(* CoDeSys 2.3.9.41 project: VOS_Vorkuta_ASU_3_osmos_2.pro *)
(* Libraries: PID_Regulators.lib 6.11.19 15:29:27, Util.lib 18.5.10 15:14:28, STANDARD.LIB 4.10.05 11:14:46, IECSFC.LIB 13.4.06 15:51:28, GermesLib_1_4.lib 25.4.21 16:11:00, SYSLIBTIME.LIB 6.11.19 15:29:28, ANALYZATION.LIB 5.10.99 09:05:06 *)

(* PLC configuration (modules and I/O channels)
Fast discrete inputs [I_SIMPLE_INPUT] node 0, in %IB0 out %QB0 {ChannellName = Fast discrete inputs; Filtrationtime = 10000}
  DD1_DI_1 AT %IX0.0 [BitInput] Авария насоса Р03.01/01 {ChannellName = Enter name}
  DD1_DI_2 AT %IX0.1 [BitInput] Авария насоса Р03.01/02 {ChannellName = Enter name}
  DD1_DI_3 AT %IX0.2 [BitInput] эк.манометр PIS03.01/01 после насоса Р03.01/01 {ChannellName = Enter name}
  DD1_DI_4 AT %IX0.3 [BitInput] эк.манометр PIS03.01/02 после насоса Р03.01/02 {ChannellName = Enter name}
Discrete inputs [ID130] node 1, in %IB1 out %QB1 {ChannellName = Discrete inputs; Filtrationtime_GeneralINP = 10; PinCount = 12; Visibility = No}
  AT %IB1.0 [ByteInput] 8 discrete inputs {ChannellName = Enter name}
  AT %IB1.1 [ByteInput] 4 discrete inputs {ChannellName = Enter name}
Fast discrete outputs [OWEN_ID570] node 2, in %IB2 out %QB2 {ChannellName = Fast discrete outputs; SafeValueBool = FALSE; SafeValueBool = FALSE; SafeValueBool = FALSE; SafeValueBool = FALSE; Visibility = No}
  DD1_DO_1 AT %QX2.0 [BitOutput] Fast discrete output 1 {ChannellName = Enter name}
  DD1_DO_2 AT %QX2.1 [BitOutput] Fast discrete output 2 {ChannellName = Enter name}
  DD1_DO_3 AT %QX2.2 [BitOutput] Fast discrete output 3 {ChannellName = Enter name}
  DD1_DO_4 AT %QX2.3 [BitOutput] Fast discrete output 4 {ChannellName = Enter name}
Discrete outputs [ID131] node 3, in %IB3 out %QB3 {ChannellName = Discrete outputs; SafeValueByte = 0; Visibility = No}
  AT %QB3.0 [ByteOutput] 8 discrete outputs {ChannellName = Enter name}
  AT %QB3.1 [ByteOutput] 8 discrete outputs {ChannellName = Enter name}
Fast analog inputs [ID125] node 4, in %IB4 out %QB4 {ChannellName = Fast analog inputs; Flt_Comm = 50Hz 2Por}
  DD1_AI_1 AT %IR4.0 [FloatInputP] резерв {ChannellName = Fast analog input; AIN_TYPE = 0-20 mA; Peak_Filtr = 200; Flt_Ch = Off; TauRC = 10; MinFV = 0; MaxFV = 20}
  DD1_AI_2 AT %IR4.1 [FloatInputP] датчик давления РТ03.01/01 {ChannellName = Fast analog input; AIN_TYPE = 0-20 mA; Peak_Filtr = 200; Flt_Ch = Off; TauRC = 10; MinFV = 0; MaxFV = 20}
  DD1_AI_3 AT %IR4.2 [FloatInputP] датчик давления РТ03.02/01 {ChannellName = Fast analog input; AIN_TYPE = 0-20 mA; Peak_Filtr = 200; Flt_Ch = Off; TauRC = 10; MinFV = 0; MaxFV = 20}
  DD1_AI_4 AT %IR4.3 [FloatInputP] датчик давления РТ03.03/01 {ChannellName = Fast analog input; AIN_TYPE = 0-20 mA; Peak_Filtr = 200; Flt_Ch = Off; TauRC = 10; MinFV = 0; MaxFV = 20}
  DD1_AI_5 AT %IR4.4 [FloatInputP] датчик давления РТ03.04/01 {ChannellName = Fast analog input; AIN_TYPE = 0-20 mA; Peak_Filtr = 200; Flt_Ch = Off; TauRC = 10; MinFV = 0; MaxFV = 20}
  DD1_AI_6 AT %IR4.5 [FloatInputP] кондуктомер QIT03.01/01 осн.осмос {ChannellName = Fast analog input; AIN_TYPE = 0-20 mA; Peak_Filtr = 200; Flt_Ch = Off; TauRC = 10; MinFV = 0; MaxFV = 20}
  DD1_AI_7 AT %IR4.6 [FloatInputP] расходомер FIT03.02/01 осн.осмос {ChannellName = Fast analog input; AIN_TYPE = 0-20 mA; Peak_Filtr = 200; Flt_Ch = Off; TauRC = 10; MinFV = 0; MaxFV = 20}
  DD1_AI_8 AT %IR4.7 [FloatInputP] расходомер FIT03.03/01 осн.осмос {ChannellName = Fast analog input; AIN_TYPE = 0-20 mA; Peak_Filtr = 200; Flt_Ch = Off; TauRC = 10; MinFV = 0; MaxFV = 20}
  AT %IW4.8 [WordInput] AI read time (10ms) {ChannellName = Enter name}
Analog outputs [ID126] node 5, in %IB5 out %QB5 {ChannellName = Analog outputs}
  DD1_AO_1 AT %QR5.0 [FloatOutputP] производительность осн.доз.насоса Р03.02/01 {ChannellName = Analog output; AOUT_TYPE = 4-20 mA; SafeValueREAL = 0.0}
  DD1_AO_2 AT %QR5.1 [FloatOutputP] производительность рез.доз.насоса Р03.02/02 {ChannellName = Analog output; AOUT_TYPE = 4-20 mA; SafeValueREAL = 0.0}
  DD1_AO_3 AT %QR5.2 [FloatOutputP] резерв {ChannellName = Analog output; AOUT_TYPE = 4-20 mA; SafeValueREAL = 0.0}
  DD1_AO_4 AT %QR5.3 [FloatOutputP] резерв {ChannellName = Analog output; AOUT_TYPE = 4-20 mA; SafeValueREAL = 0.0}
Special input [ID103] node 6, in %IB6 out %QB6 {ChannellName = Special input}
  AT %IX6.0 [BitInput] Special input {ChannellName = Enter name}
Special output [ID104] node 7, in %IB7 out %QB7 {ChannellName = Special output}
  AT %QX7.0 [BitOutput] Special output {ChannellName = Enter name}
ModBus (Master) [MODBUS_MASTER_ID450] node 8, in %IB8 out %QB8 {ChannellName = ModBus (Master); Visibility = No}
  AT %QD8.0 [DWordOutput] Last address {ChannellName = Enter name}
  AT %QW8.1 [WordOutput] Last error {ChannellName = Enter name}
  RS-485-1 [COM1_USART] node 0, in %IB8.0 out %QB8.0 {ChannellName = RS-485-1; CommunicationSpeed = 9600; Parity = NO PARITY CHECK; BitLength = 8 bits; StopLength = One stop bit; InterfaceType = RS485; FrameOriented = RTU; Timeout = 5; Visibility = No}
  Universal Modbus device [ID2000] node 1, in %IB8.1 out %QB8.1 {ChannellName = Universal Modbus device; ModuleIP = 10:0:0:223; ServiceTimeout = 150; TCPport = 502; NetMode = Serial; ModuleSlaveAddress = 11; RequestType = By poll time; PeriodOfService = 100; Visibility = No; RepeatCounter = 0; ByteSequence = Native}
    AT %QB8.1.0 [ComChannel] Command (0xff - Start) {ChannellName = Enter name}
    Real input module [ID2007] node 0, in %IB8.1.0 out %QB8.1.0 {ChannellName = float input module; ModbusAddress = 512; Command_read_regs = Read holding Registers  (0x03); Visibility = No}
      PT030102rawValue AT %QD8.1.0.0 [FloatOutput] {ChannellName = Enter name}
    Real input module [ID2007] node 1, in %IB8.1.1 out %QB8.1.1 {ChannellName = float input module; ModbusAddress = 514; Command_read_regs = Read holding Registers  (0x03); Visibility = No}
      PT030202rawValue AT %QD8.1.1.0 [FloatOutput] {ChannellName = Enter name}
    Real input module [ID2007] node 2, in %IB8.1.2 out %QB8.1.2 {ChannellName = float input module; ModbusAddress = 516; Command_read_regs = Read holding Registers  (0x03); Visibility = No}
      PT030302rawValue AT %QD8.1.2.0 [FloatOutput] {ChannellName = Enter name}
    Real input module [ID2007] node 3, in %IB8.1.3 out %QB8.1.3 {ChannellName = float input module; ModbusAddress = 518; Command_read_regs = Read holding Registers  (0x03); Visibility = No}
      PT030402rawValue AT %QD8.1.3.0 [FloatOutput] {ChannellName = Enter name}
    Real input module [ID2007] node 4, in %IB8.1.4 out %QB8.1.4 {ChannellName = float input module; ModbusAddress = 520; Command_read_regs = Read holding Registers  (0x03); Visibility = No}
      QIT030102rawValue AT %QD8.1.4.0 [FloatOutput] {ChannellName = Enter name}
    Real input module [ID2007] node 5, in %IB8.1.5 out %QB8.1.5 {ChannellName = float input module; ModbusAddress = 522; Command_read_regs = Read holding Registers  (0x03); Visibility = No}
      FIT030202rawValue AT %QD8.1.5.0 [FloatOutput] {ChannellName = Enter name}
    Real input module [ID2007] node 6, in %IB8.1.6 out %QB8.1.6 {ChannellName = float input module; ModbusAddress = 524; Command_read_regs = Read holding Registers  (0x03); Visibility = No}
      FIT030302rawValue AT %QD8.1.6.0 [FloatOutput] {ChannellName = Enter name}
    Real input module [ID2007] node 7, in %IB8.1.7 out %QB8.1.7 {ChannellName = float input module; ModbusAddress = 526; Command_read_regs = Read holding Registers  (0x03); Visibility = No}
      FIT030101rawValue AT %QD8.1.7.0 [FloatOutput] {ChannellName = Enter name}
    Register input module [ID2003] node 8, in %IB8.1.8 out %QB8.1.8 {ChannellName = Register input module; ModbusAddress = 529; Command_read_regs = Read input registers  (0x04); Visibility = No}
      DI_bit_mask_DD2 AT %QW8.1.8.0 [WordOutput] {ChannellName = Enter name}
    Register input module [ID2003] node 9, in %IB8.1.9 out %QB8.1.9 {ChannellName = Register input module; ModbusAddress = 532; Command_read_regs = Read input registers  (0x04); Visibility = No}
      stat_word_P030601_PLC AT %QW8.1.9.0 [WordOutput] {ChannellName = Enter name}
    Register input module [ID2003] node 10, in %IB8.1.10 out %QB8.1.10 {ChannellName = Register input module; ModbusAddress = 535; Command_read_regs = Read input registers  (0x04); Visibility = No}
      stat_word_P030602_PLC AT %QW8.1.10.0 [WordOutput] {ChannellName = Enter name}
  Universal Modbus device [ID2000] node 2, in %IB8.2 out %QB8.2 {ChannellName = Universal Modbus device; ModuleIP = 10:0:0:223; ServiceTimeout = 150; TCPport = 502; NetMode = Serial; ModuleSlaveAddress = 1; RequestType = By value change; PeriodOfService = 100; Visibility = No; RepeatCounter = 0; ByteSequence = Native}
    AT %QB8.2.0 [ComChannel] Command (0xff - Start) {ChannellName = Enter name}
    Register output module [ID2004] node 0, in %IB8.2.0 out %QB8.2.0 {ChannellName = Register; ModbusAddress = 528; Command_write_one_reg = Write multiple registers(0x10); Visibility = No}
      DO_bit_mask_DD2 AT %QW8.2.0.0 [WordOutput] {ChannellName = Enter name}
    Register output module [ID2004] node 1, in %IB8.2.1 out %QB8.2.1 {ChannellName = Register; ModbusAddress = 530; Command_write_one_reg = Write multiple registers(0x10); Visibility = No}
      com_word_P030601_PLC AT %QW8.2.1.0 [WordOutput] {ChannellName = Enter name}
    Register output module [ID2004] node 2, in %IB8.2.2 out %QB8.2.2 {ChannellName = Register; ModbusAddress = 531; Command_write_one_reg = Write multiple registers(0x10); Visibility = No}
      set_freq_P030601_PLC AT %QW8.2.2.0 [WordOutput] {ChannellName = Enter name}
    Register output module [ID2004] node 3, in %IB8.2.3 out %QB8.2.3 {ChannellName = Register; ModbusAddress = 533; Command_write_one_reg = Write multiple registers(0x10); Visibility = No}
      com_word_P030602_PLC AT %QW8.2.3.0 [WordOutput] {ChannellName = Enter name}
    Register output module [ID2004] node 4, in %IB8.2.4 out %QB8.2.4 {ChannellName = Register; ModbusAddress = 534; Command_write_one_reg = Write multiple registers(0x10); Visibility = No}
      set_freq_P030602_PLC AT %QW8.2.4.0 [WordOutput] {ChannellName = Enter name}
ModBus (Master) [MODBUS_MASTER_ID450] node 9, in %IB9 out %QB9 {ChannellName = ModBus (Master); Visibility = No}
  AT %QD9.0 [DWordOutput] Last address {ChannellName = Enter name}
  AT %QW9.1 [WordOutput] Last error {ChannellName = Enter name}
  RS-232 [COM2_USART] node 0, in %IB9.0 out %QB9.0 {ChannellName = RS-232; CommunicationSpeed = 115200; Parity = NO PARITY CHECK; BitLength = 8 bits; StopLength = One stop bit; InterfaceType = RS232; FrameOriented = RTU; Timeout = 5; Visibility = No}
  Universal Modbus device [ID2000] node 1, in %IB9.1 out %QB9.1 {ChannellName = Universal Modbus device; ModuleIP = 10:0:0:223; ServiceTimeout = 150; TCPport = 502; NetMode = Serial; ModuleSlaveAddress = 1; RequestType = By poll time; PeriodOfService = 50; Visibility = No; RepeatCounter = 0; ByteSequence = Native}
    AT %QB9.1.0 [ComChannel] Command (0xff - Start) {ChannellName = Enter name}
    Register input module [ID2003] node 0, in %IB9.1.0 out %QB9.1.0 {ChannellName = Register input module; ModbusAddress = 10256; Command_read_regs = Read holding Registers  (0x03); Visibility = No}
      PANsetWordP0301 AT %QW9.1.0.0 [WordOutput] {ChannellName = Enter name}
    Register input module [ID2003] node 1, in %IB9.1.1 out %QB9.1.1 {ChannellName = Register input module; ModbusAddress = 10257; Command_read_regs = Read holding Registers  (0x03); Visibility = No}
      PANsetWordP0302 AT %QW9.1.1.0 [WordOutput] {ChannellName = Enter name}
PAN_FIT0301maxValue AT %QD9.1.2.0 [FloatOutput] {ChannellName = Enter name}
Real input module [ID2007] node 3, in %IB9.1.3 out %QB9.1.3 {ChannellName = float input module; ModbusAddress = 10260; Command_read_regs = Read holding Registers  (0x03); Visibility = No}
  PANsetMaxPumpDosingValueP0302 AT %QD9.1.3.0 [FloatOutput] {ChannellName = Enter name}
Real input module [ID2007] node 4, in %IB9.1.4 out %QB9.1.4 {ChannellName = float input module; ModbusAddress = 10262; Command_read_regs = Read holding Registers  (0x03); Visibility = No}
  PANsetKoeffPropotrionalityP0302 AT %QD9.1.4.0 [FloatOutput] {ChannellName = Enter name}
Register input module [ID2003] node 5, in %IB9.1.5 out %QB9.1.5 {ChannellName = Register input module; ModbusAddress = 10264; Command_read_regs = Read holding Registers  (0x03); Visibility = No}
  PAN_CHECKING_DELAY_TIME AT %QW9.1.5.0 [WordOutput] {ChannellName = Enter name}
Register input module [ID2003] node 6, in %IB9.1.6 out %QB9.1.6 {ChannellName = Register input module; ModbusAddress = 10265; Command_read_regs = Read holding Registers  (0x03); Visibility = No}
  PAN_DELAY_REPEATED_START_SEC AT %QW9.1.6.0 [WordOutput] {ChannellName = Enter name}
Register input module [ID2003] node 7, in %IB9.1.7 out %QB9.1.7 {ChannellName = Register input module; ModbusAddress = 10266; Command_read_regs = Read holding Registers  (0x03); Visibility = No}
  PAN_DELAY_TO_OFF_VALVE AT %QW9.1.7.0 [WordOutput] {ChannellName = Enter name}
Register input module [ID2003] node 8, in %IB9.1.8 out %QB9.1.8 {ChannellName = Register input module; ModbusAddress = 10267; Command_read_regs = Read holding Registers  (0x03); Visibility = No}
  PAN_DELAY_TO_CHECK_PT0301 AT %QW9.1.8.0 [WordOutput] {ChannellName = Enter name}
Register input module [ID2003] node 9, in %IB9.1.9 out %QB9.1.9 {ChannellName = Register input module; ModbusAddress = 10268; Command_read_regs = Read holding Registers  (0x03); Visibility = No}
  PAN_DELAY_TO_SWITCH_VALVE AT %QW9.1.9.0 [WordOutput] {ChannellName = Enter name}
Register input module [ID2003] node 10, in %IB9.1.10 out %QB9.1.10 {ChannellName = Register input module; ModbusAddress = 10269; Command_read_regs = Read holding Registers  (0x03); Visibility = No}
  PAN_DELAY_TO_CLOSE_VALVE AT %QW9.1.10.0 [WordOutput] {ChannellName = Enter name}
Real input module [ID2007] node 11, in %IB9.1.11 out %QB9.1.11 {ChannellName = float input module; ModbusAddress = 10276; Command_read_regs = Read holding Registers  (0x03); Visibility = No}
  PAN_FIT030201maxValue AT %QD9.1.11.0 [FloatOutput] {ChannellName = Enter name}
Real input module [ID2007] node 12, in %IB9.1.12 out %QB9.1.12 {ChannellName = float input module; ModbusAddress = 10278; Command_read_regs = Read holding Registers  (0x03); Visibility = No}
  PAN_FIT030301maxValue AT %QD9.1.12.0 [FloatOutput] {ChannellName = Enter name}
Real input module [ID2007] node 13, in %IB9.1.13 out %QB9.1.13 {ChannellName = float input module; ModbusAddress = 10280; Command_read_regs = Read holding Registers  (0x03); Visibility = No}
  PAN_FIT030202maxValue AT %QD9.1.13.0 [FloatOutput] {ChannellName = Enter name}
Real input module [ID2007] node 14, in %IB9.1.14 out %QB9.1.14 {ChannellName = float input module; ModbusAddress = 10282; Command_read_regs = Read holding Registers  (0x03); Visibility = No}
  PAN_FIT030302maxValue AT %QD9.1.14.0 [FloatOutput] {ChannellName = Enter name}
Real input module [ID2007] node 15, in %IB9.1.15 out %QB9.1.15 {ChannellName = float input module; ModbusAddress = 10284; Command_read_regs = Read holding Registers  (0x03); Visibility = No}
  PAN_QIT030101maxValue AT %QD9.1.15.0 [FloatOutput] {ChannellName = Enter name}
Real input module [ID2007] node 16, in %IB9.1.16 out %QB9.1.16 {ChannellName = float input module; ModbusAddress = 10286; Command_read_regs = Read holding Registers  (0x03); Visibility = No}
  PAN_QIT030102maxValue AT %QD9.1.16.0 [FloatOutput] {ChannellName = Enter name}
Real input module [ID2007] node 17, in %IB9.1.17 out %QB9.1.17 {ChannellName = float input module; ModbusAddress = 10288; Command_read_regs = Read holding Registers  (0x03); Visibility = No}
  PAN_PT030101maxValue AT %QD9.1.17.0 [FloatOutput] {ChannellName = Enter name}
Real input module [ID2007] node 18, in %IB9.1.18 out %QB9.1.18 {ChannellName = float input module; ModbusAddress = 10290; Command_read_regs = Read holding Registers  (0x03); Visibility = No}
  PAN_PT030201maxValue AT %QD9.1.18.0 [FloatOutput] {ChannellName = Enter name}
Real input module [ID2007] node 19, in %IB9.1.19 out %QB9.1.19 {ChannellName = float input module; ModbusAddress = 10292; Command_read_regs = Read holding Registers  (0x03); Visibility = No}
  PAN_PT030301maxValue AT %QD9.1.19.0 [FloatOutput] {ChannellName = Enter name}
Real input module [ID2007] node 20, in %IB9.1.20 out %QB9.1.20 {ChannellName = float input module; ModbusAddress = 10294; Command_read_regs = Read holding Registers  (0x03); Visibility = No}
  PAN_PT030401maxValue AT %QD9.1.20.0 [FloatOutput] {ChannellName = Enter name}
Real input module [ID2007] node 21, in %IB9.1.21 out %QB9.1.21 {ChannellName = float input module; ModbusAddress = 10296; Command_read_regs = Read holding Registers  (0x03); Visibility = No}
  PAN_PT030102maxValue AT %QD9.1.21.0 [FloatOutput] {ChannellName = Enter name}
Real input module [ID2007] node 22, in %IB9.1.22 out %QB9.1.22 {ChannellName = float input module; ModbusAddress = 10298; Command_read_regs = Read holding Registers  (0x03); Visibility = No}
  PAN_PT030202maxValue AT %QD9.1.22.0 [FloatOutput] {ChannellName = Enter name}
Real input module [ID2007] node 23, in %IB9.1.23 out %QB9.1.23 {ChannellName = float input module; ModbusAddress = 10300; Command_read_regs = Read holding Registers  (0x03); Visibility = No}
  PAN_PT030302maxValue AT %QD9.1.23.0 [FloatOutput] {ChannellName = Enter name}
Real input module [ID2007] node 24, in %IB9.1.24 out %QB9.1.24 {ChannellName = float input module; ModbusAddress = 10302; Command_read_regs = Read holding Registers  (0x03); Visibility = No}
  PAN_PT030402maxValue AT %QD9.1.24.0 [FloatOutput] {ChannellName = Enter name}
PANsetWordOsmos AT %QW9.1.25.0 [WordOutput] {ChannellName = Enter name}
Real input module [ID2007] node 26, in %IB9.1.26 out %QB9.1.26 {ChannellName = float input module; ModbusAddress = 10306; Command_read_regs = Read holding Registers  (0x03); Visibility = No}
  PAN_PT0301startValue AT %QD9.1.26.0 [FloatOutput] {ChannellName = Enter name}
Real input module [ID2007] node 27, in %IB9.1.27 out %QB9.1.27 {ChannellName = float input module; ModbusAddress = 10308; Command_read_regs = Read holding Registers  (0x03); Visibility = No}
  PAN_FIT0303setValue AT %QD9.1.27.0 [FloatOutput] {ChannellName = Enter name}
Real input module [ID2007] node 28, in %IB9.1.28 out %QB9.1.28 {ChannellName = float input module; ModbusAddress = 10310; Command_read_regs = Read holding Registers  (0x03); Visibility = No}
  PAN_PT0302setMaxValue AT %QD9.1.28.0 [FloatOutput] {ChannellName = Enter name}
Real input module [ID2007] node 29, in %IB9.1.29 out %QB9.1.29 {ChannellName = float input module; ModbusAddress = 10312; Command_read_regs = Read holding Registers  (0x03); Visibility = No}
  PAN_PT0303setMaxValue AT %QD9.1.29.0 [FloatOutput] {ChannellName = Enter name}
Real input module [ID2007] node 30, in %IB9.1.30 out %QB9.1.30 {ChannellName = float input module; ModbusAddress = 10314; Command_read_regs = Read holding Registers  (0x03); Visibility = No}
  PAN_PT0304setMaxValue AT %QD9.1.30.0 [FloatOutput] {ChannellName = Enter name}
Real input module [ID2007] node 31, in %IB9.1.31 out %QB9.1.31 {ChannellName = float input module; ModbusAddress = 10316; Command_read_regs = Read holding Registers  (0x03); Visibility = No}
  PAN_KP_F_P030601 AT %QD9.1.31.0 [FloatOutput] {ChannellName = Enter name}
Real input module [ID2007] node 32, in %IB9.1.32 out %QB9.1.32 {ChannellName = float input module; ModbusAddress = 10318; Command_read_regs = Read holding Registers  (0x03); Visibility = No}
  PAN_I_F_P030601 AT %QD9.1.32.0 [FloatOutput] {ChannellName = Enter name}
Real input module [ID2007] node 33, in %IB9.1.33 out %QB9.1.33 {ChannellName = float input module; ModbusAddress = 10320; Command_read_regs = Read holding Registers  (0x03); Visibility = No}
  PAN_D_F_P030601 AT %QD9.1.33.0 [FloatOutput] {ChannellName = Enter name}
Real input module [ID2007] node 34, in %IB9.1.34 out %QB9.1.34 {ChannellName = float input module; ModbusAddress = 10322; Command_read_regs = Read holding Registers  (0x03); Visibility = No}
  PAN_KP_P_P030601 AT %QD9.1.34.0 [FloatOutput] {ChannellName = Enter name}
Real input module [ID2007] node 35, in %IB9.1.35 out %QB9.1.35 {ChannellName = float input module; ModbusAddress = 10324; Command_read_regs = Read holding Registers  (0x03); Visibility = No}
  PAN_I_P_P030601 AT %QD9.1.35.0 [FloatOutput] {ChannellName = Enter name}
Real input module [ID2007] node 36, in %IB9.1.36 out %QB9.1.36 {ChannellName = float input module; ModbusAddress = 10326; Command_read_regs = Read holding Registers  (0x03); Visibility = No}
  PAN_D_P_P030601 AT %QD9.1.36.0 [FloatOutput] {ChannellName = Enter name}
Real input module [ID2007] node 37, in %IB9.1.37 out %QB9.1.37 {ChannellName = float input module; ModbusAddress = 10328; Command_read_regs = Read holding Registers  (0x03); Visibility = No}
  PAN_KP_F_P030602 AT %QD9.1.37.0 [FloatOutput] {ChannellName = Enter name}
Real input module [ID2007] node 38, in %IB9.1.38 out %QB9.1.38 {ChannellName = float input module; ModbusAddress = 10330; Command_read_regs = Read holding Registers  (0x03); Visibility = No}
  PAN_I_F_P030602 AT %QD9.1.38.0 [FloatOutput] {ChannellName = Enter name}
Real input module [ID2007] node 39, in %IB9.1.39 out %QB9.1.39 {ChannellName = float input module; ModbusAddress = 10332; Command_read_regs = Read holding Registers  (0x03); Visibility = No}
  PAN_D_F_P030602 AT %QD9.1.39.0 [FloatOutput] {ChannellName = Enter name}
Real input module [ID2007] node 40, in %IB9.1.40 out %QB9.1.40 {ChannellName = float input module; ModbusAddress = 10334; Command_read_regs = Read holding Registers  (0x03); Visibility = No}
  PAN_KP_P_P030602 AT %QD9.1.40.0 [FloatOutput] {ChannellName = Enter name}
Real input module [ID2007] node 41, in %IB9.1.41 out %QB9.1.41 {ChannellName = float input module; ModbusAddress = 10336; Command_read_regs = Read holding Registers  (0x03); Visibility = No}
  PAN_I_P_P030602 AT %QD9.1.41.0 [FloatOutput] {ChannellName = Enter name}
Real input module [ID2007] node 42, in %IB9.1.42 out %QB9.1.42 {ChannellName = float input module; ModbusAddress = 10338; Command_read_regs = Read holding Registers  (0x03); Visibility = No}
  PAN_D_P_P030602 AT %QD9.1.42.0 [FloatOutput] {ChannellName = Enter name}
  PAN_FIT0303_SetCascade AT %QD9.1.43.0 [FloatOutput] {ChannellName = Enter name}
ID2003NoNoINTRegister input module, AT %QW9.1.44.0 [WordOutput] B	,%QB	,%MB	,%MPAN_valuesActivator {ChannellName = Enter name}
Universal Modbus device [ID2000] node 2, in %IB9.2 out %QB9.2 {ChannellName = Universal Modbus device; ModuleIP = 10:0:0:223; ServiceTimeout = 150; TCPport = 502; NetMode = Serial; ModuleSlaveAddress = 1; RequestType = Both; PeriodOfService = 100; Visibility = No; RepeatCounter = 0; ByteSequence = Native}
  AT %QB9.2.0 [ComChannel] Command (0xff - Start) {ChannellName = Enter name}
  Register output module [ID2004] node 0, in %IB9.2.0 out %QB9.2.0 {ChannellName = Register; ModbusAddress = 256; Command_write_one_reg = Write multiple registers(0x10); Visibility = No}
    PANstatWordP0301 AT %QW9.2.0.0 [WordOutput] {ChannellName = Enter name}
  Register output module [ID2004] node 1, in %IB9.2.1 out %QB9.2.1 {ChannellName = Register; ModbusAddress = 257; Command_write_one_reg = Write multiple registers(0x10); Visibility = No}
    PANdaysOfWorkP030101 AT %QW9.2.1.0 [WordOutput] {ChannellName = Enter name}
  Register output module [ID2004] node 2, in %IB9.2.2 out %QB9.2.2 {ChannellName = Register; ModbusAddress = 258; Command_write_one_reg = Write multiple registers(0x10); Visibility = No}
    PANhoursOfWorkP030101 AT %QW9.2.2.0 [WordOutput] {ChannellName = Enter name}
  Register output module [ID2004] node 3, in %IB9.2.3 out %QB9.2.3 {ChannellName = Register; ModbusAddress = 259; Command_write_one_reg = Write multiple registers(0x10); Visibility = No}
    PANminutesOfWorkP030101 AT %QW9.2.3.0 [WordOutput] {ChannellName = Enter name}
  Register output module [ID2004] node 4, in %IB9.2.4 out %QB9.2.4 {ChannellName = Register; ModbusAddress = 260; Command_write_one_reg = Write multiple registers(0x10); Visibility = No}
    PANsecondsOfWorkP030101 AT %QW9.2.4.0 [WordOutput] {ChannellName = Enter name}
  Register output module [ID2004] node 5, in %IB9.2.5 out %QB9.2.5 {ChannellName = Register; ModbusAddress = 261; Command_write_one_reg = Write multiple registers(0x10); Visibility = No}
    PANtoNextStartP030101timer AT %QW9.2.5.0 [WordOutput] {ChannellName = Enter name}
  Real output module [ID2008] node 6, in %IB9.2.6 out %QB9.2.6 {ChannellName = float output module; ModbusAddress = 262; Command_write_regs = Preset multiple Registers (0x10); Visibility = No}
    PANcounterP030101 AT %QD9.2.6.0 [FloatOutput] {ChannellName = Enter name}
  Real output module [ID2008] node 7, in %IB9.2.7 out %QB9.2.7 {ChannellName = float output module; ModbusAddress = 264; Command_write_regs = Preset multiple Registers (0x10); Visibility = No}
    PANcounterP030102 AT %QD9.2.7.0 [FloatOutput] {ChannellName = Enter name}
  Register output module [ID2004] node 8, in %IB9.2.8 out %QB9.2.8 {ChannellName = Register; ModbusAddress = 266; Command_write_one_reg = Write multiple registers(0x10); Visibility = No}
    PANdaysOfWorkP030102 AT %QW9.2.8.0 [WordOutput] {ChannellName = Enter name}
  Register output module [ID2004] node 9, in %IB9.2.9 out %QB9.2.9 {ChannellName = Register; ModbusAddress = 267; Command_write_one_reg = Write multiple registers(0x10); Visibility = No}
    PANhoursOfWorkP030102 AT %QW9.2.9.0 [WordOutput] {ChannellName = Enter name}
  Register output module [ID2004] node 10, in %IB9.2.10 out %QB9.2.10 {ChannellName = Register; ModbusAddress = 268; Command_write_one_reg = Write multiple registers(0x10); Visibility = No}
    PANminutesOfWorkP030102 AT %QW9.2.10.0 [WordOutput] {ChannellName = Enter name}
  Register output module [ID2004] node 11, in %IB9.2.11 out %QB9.2.11 {ChannellName = Register; ModbusAddress = 269; Command_write_one_reg = Write multiple registers(0x10); Visibility = No}
    PANsecondsOfWorkP030102 AT %QW9.2.11.0 [WordOutput] {ChannellName = Enter name}
  Register output module [ID2004] node 12, in %IB9.2.12 out %QB9.2.12 {ChannellName = Register; ModbusAddress = 270; Command_write_one_reg = Write multiple registers(0x10); Visibility = No}
    PANtoNextStartP030102timer AT %QW9.2.12.0 [WordOutput] {ChannellName = Enter name}
  Register output module [ID2004] node 13, in %IB9.2.13 out %QB9.2.13 {ChannellName = Register; ModbusAddress = 271; Command_write_one_reg = Write multiple registers(0x10); Visibility = No}
    PANstatWordP0302 AT %QW9.2.13.0 [WordOutput] {ChannellName = Enter name}
  Register output module [ID2004] node 14, in %IB9.2.14 out %QB9.2.14 {ChannellName = Register; ModbusAddress = 272; Command_write_one_reg = Write multiple registers(0x10); Visibility = No}
    PANdaysOfWorkP030201 AT %QW9.2.14.0 [WordOutput] {ChannellName = Enter name}
  Register output module [ID2004] node 15, in %IB9.2.15 out %QB9.2.15 {ChannellName = Register; ModbusAddress = 273; Command_write_one_reg = Write multiple registers(0x10); Visibility = No}
    PANhoursOfWorkP030201 AT %QW9.2.15.0 [WordOutput] {ChannellName = Enter name}
  Register output module [ID2004] node 16, in %IB9.2.16 out %QB9.2.16 {ChannellName = Register; ModbusAddress = 274; Command_write_one_reg = Write multiple registers(0x10); Visibility = No}
    PANminutesOfWorkP030201 AT %QW9.2.16.0 [WordOutput] {ChannellName = Enter name}
  Register output module [ID2004] node 17, in %IB9.2.17 out %QB9.2.17 {ChannellName = Register; ModbusAddress = 275; Command_write_one_reg = Write multiple registers(0x10); Visibility = No}
    PANsecondsOfWorkP030201 AT %QW9.2.17.0 [WordOutput] {ChannellName = Enter name}
  Register output module [ID2004] node 18, in %IB9.2.18 out %QB9.2.18 {ChannellName = Register; ModbusAddress = 276; Command_write_one_reg = Write multiple registers(0x10); Visibility = No}
    PANtoNextStartP030201timer AT %QW9.2.18.0 [WordOutput] {ChannellName = Enter name}
  Register output module [ID2004] node 19, in %IB9.2.19 out %QB9.2.19 {ChannellName = Register; ModbusAddress = 277; Command_write_one_reg = Write multiple registers(0x10); Visibility = No}
    PANdaysOfWorkP030202 AT %QW9.2.19.0 [WordOutput] {ChannellName = Enter name}
  Register output module [ID2004] node 20, in %IB9.2.20 out %QB9.2.20 {ChannellName = Register; ModbusAddress = 278; Command_write_one_reg = Write multiple registers(0x10); Visibility = No}
    PANhoursOfWorkP030202 AT %QW9.2.20.0 [WordOutput] {ChannellName = Enter name}
  Register output module [ID2004] node 21, in %IB9.2.21 out %QB9.2.21 {ChannellName = Register; ModbusAddress = 279; Command_write_one_reg = Write multiple registers(0x10); Visibility = No}
    PANminutesOfWorkP030202 AT %QW9.2.21.0 [WordOutput] {ChannellName = Enter name}
  Register output module [ID2004] node 22, in %IB9.2.22 out %QB9.2.22 {ChannellName = Register; ModbusAddress = 280; Command_write_one_reg = Write multiple registers(0x10); Visibility = No}
    PANsecondsOfWorkP030202 AT %QW9.2.22.0 [WordOutput] {ChannellName = Enter name}
  Register output module [ID2004] node 23, in %IB9.2.23 out %QB9.2.23 {ChannellName = Register; ModbusAddress = 281; Command_write_one_reg = Write multiple registers(0x10); Visibility = No}
    PANtoNextStartP030202timer AT %QW9.2.23.0 [WordOutput] {ChannellName = Enter name}
  Real output module [ID2008] node 24, in %IB9.2.24 out %QB9.2.24 {ChannellName = float output module; ModbusAddress = 282; Command_write_regs = Preset multiple Registers (0x10); Visibility = No}
    PANcounterP030201 AT %QD9.2.24.0 [FloatOutput] {ChannellName = Enter name}
  Real output module [ID2008] node 25, in %IB9.2.25 out %QB9.2.25 {ChannellName = float output module; ModbusAddress = 284; Command_write_regs = Preset multiple Registers (0x10); Visibility = No}
    PANcounterP030202 AT %QD9.2.25.0 [FloatOutput] {ChannellName = Enter name}
  Real output module [ID2008] node 26, in %IB9.2.26 out %QB9.2.26 {ChannellName = float output module; ModbusAddress = 286; Command_write_regs = Preset multiple Registers (0x10); Visibility = No}
    PAN_FIT0301realValue AT %QD9.2.26.0 [FloatOutput] {ChannellName = Enter name}
  Real output module [ID2008] node 27, in %IB9.2.27 out %QB9.2.27 {ChannellName = float output module; ModbusAddress = 288; Command_write_regs = Preset multiple Registers (0x10); Visibility = No}
    PAN_PT030101realValue AT %QD9.2.27.0 [FloatOutput] {ChannellName = Enter name}
  Real output module [ID2008] node 28, in %IB9.2.28 out %QB9.2.28 {ChannellName = float output module; ModbusAddress = 290; Command_write_regs = Preset multiple Registers (0x10); Visibility = No}
    PAN_PT030201realValue AT %QD9.2.28.0 [FloatOutput] {ChannellName = Enter name}
  Real output module [ID2008] node 29, in %IB9.2.29 out %QB9.2.29 {ChannellName = float output module; ModbusAddress = 292; Command_write_regs = Preset multiple Registers (0x10); Visibility = No}
    PAN_PT030301realValue AT %QD9.2.29.0 [FloatOutput] {ChannellName = Enter name}
  Real output module [ID2008] node 30, in %IB9.2.30 out %QB9.2.30 {ChannellName = float output module; ModbusAddress = 294; Command_write_regs = Preset multiple Registers (0x10); Visibility = No}
    PAN_FIT030301realValue AT %QD9.2.30.0 [FloatOutput] {ChannellName = Enter name}
  Real output module [ID2008] node 31, in %IB9.2.31 out %QB9.2.31 {ChannellName = float output module; ModbusAddress = 296; Command_write_regs = Preset multiple Registers (0x10); Visibility = No}
    PAN_PT030102realValue AT %QD9.2.31.0 [FloatOutput] {ChannellName = Enter name}
  Real output module [ID2008] node 32, in %IB9.2.32 out %QB9.2.32 {ChannellName = float output module; ModbusAddress = 298; Command_write_regs = Preset multiple Registers (0x10); Visibility = No}
    PAN_PT030202realValue AT %QD9.2.32.0 [FloatOutput] {ChannellName = Enter name}
  Real output module [ID2008] node 33, in %IB9.2.33 out %QB9.2.33 {ChannellName = float output module; ModbusAddress = 300; Command_write_regs = Preset multiple Registers (0x10); Visibility = No}
    PAN_PT030302realValue AT %QD9.2.33.0 [FloatOutput] {ChannellName = Enter name}
  Real output module [ID2008] node 34, in %IB9.2.34 out %QB9.2.34 {ChannellName = float output module; ModbusAddress = 302; Command_write_regs = Preset multiple Registers (0x10); Visibility = No}
    PAN_FIT030302realValue AT %QD9.2.34.0 [FloatOutput] {ChannellName = Enter name}
  Real output module [ID2008] node 35, in %IB9.2.35 out %QB9.2.35 {ChannellName = float output module; ModbusAddress = 304; Command_write_regs = Preset multiple Registers (0x10); Visibility = No}
    PAN_PT030401realValue AT %QD9.2.35.0 [FloatOutput] {ChannellName = Enter name}
  Real output module [ID2008] node 36, in %IB9.2.36 out %QB9.2.36 {ChannellName = float output module; ModbusAddress = 306; Command_write_regs = Preset multiple Registers (0x10); Visibility = No}
    PAN_FIT030201realValue AT %QD9.2.36.0 [FloatOutput] {ChannellName = Enter name}
  Real output module [ID2008] node 37, in %IB9.2.37 out %QB9.2.37 {ChannellName = float output module; ModbusAddress = 308; Command_write_regs = Preset multiple Registers (0x10); Visibility = No}
    PAN_QIT030101realValue AT %QD9.2.37.0 [FloatOutput] {ChannellName = Enter name}
  Real output module [ID2008] node 38, in %IB9.2.38 out %QB9.2.38 {ChannellName = float output module; ModbusAddress = 310; Command_write_regs = Preset multiple Registers (0x10); Visibility = No}
    PAN_PT030402realValue AT %QD9.2.38.0 [FloatOutput] {ChannellName = Enter name}
  Real output module [ID2008] node 39, in %IB9.2.39 out %QB9.2.39 {ChannellName = float output module; ModbusAddress = 312; Command_write_regs = Preset multiple Registers (0x10); Visibility = No}
    PAN_FIT030202realValue AT %QD9.2.39.0 [FloatOutput] {ChannellName = Enter name}
  Real output module [ID2008] node 40, in %IB9.2.40 out %QB9.2.40 {ChannellName = float output module; ModbusAddress = 314; Command_write_regs = Preset multiple Registers (0x10); Visibility = No}
    PAN_QIT030102realValue AT %QD9.2.40.0 [FloatOutput] {ChannellName = Enter name}
  Register output module [ID2004] node 41, in %IB9.2.41 out %QB9.2.41 {ChannellName = Register; ModbusAddress = 316; Command_write_one_reg = Write multiple registers(0x10); Visibility = No}
    PANstatWordOsmos AT %QW9.2.41.0 [WordOutput] {ChannellName = Enter name}
  Register output module [ID2004] node 42, in %IB9.2.42 out %QB9.2.42 {ChannellName = Register; ModbusAddress = 317; Command_write_one_reg = Write multiple registers(0x10); Visibility = No}
    PANdaysOfWorkOsmos1 AT %QW9.2.42.0 [WordOutput] {ChannellName = Enter name}
  Register output module [ID2004] node 43, in %IB9.2.43 out %QB9.2.43 {ChannellName = Register; ModbusAddress = 318; Command_write_one_reg = Write multiple registers(0x10); Visibility = No}
    PANhoursOfWorkOsmos1 AT %QW9.2.43.0 [WordOutput] {ChannellName = Enter name}
  Register output module [ID2004] node 44, in %IB9.2.44 out %QB9.2.44 {ChannellName = Register; ModbusAddress = 319; Command_write_one_reg = Write multiple registers(0x10); Visibility = No}
    PANminutesOfWorkOsmos1 AT %QW9.2.44.0 [WordOutput] {ChannellName = Enter name}
  Register output module [ID2004] node 45, in %IB9.2.45 out %QB9.2.45 {ChannellName = Register; ModbusAddress = 320; Command_write_one_reg = Write multiple registers(0x10); Visibility = No}
    PANsecondsOfWorkOsmos1 AT %QW9.2.45.0 [WordOutput] {ChannellName = Enter name}
  Register output module [ID2004] node 46, in %IB9.2.46 out %QB9.2.46 {ChannellName = Register; ModbusAddress = 321; Command_write_one_reg = Write multiple registers(0x10); Visibility = No}
    PANtoNextStartOsmos1timer AT %QW9.2.46.0 [WordOutput] {ChannellName = Enter name}
  Real output module [ID2008] node 47, in %IB9.2.47 out %QB9.2.47 {ChannellName = float output module; ModbusAddress = 322; Command_write_regs = Preset multiple Registers (0x10); Visibility = No}
    PANcounterOsmos1 AT %QD9.2.47.0 [FloatOutput] {ChannellName = Enter name}
  Real output module [ID2008] node 48, in %IB9.2.48 out %QB9.2.48 {ChannellName = float output module; ModbusAddress = 324; Command_write_regs = Preset multiple Registers (0x10); Visibility = No}
    PANcounterOsmos2 AT %QD9.2.48.0 [FloatOutput] {ChannellName = Enter name}
  Register output module [ID2004] node 49, in %IB9.2.49 out %QB9.2.49 {ChannellName = Register; ModbusAddress = 326; Command_write_one_reg = Write multiple registers(0x10); Visibility = No}
    PANdaysOfWorkOsmos2 AT %QW9.2.49.0 [WordOutput] {ChannellName = Enter name}
  Register output module [ID2004] node 50, in %IB9.2.50 out %QB9.2.50 {ChannellName = Register; ModbusAddress = 327; Command_write_one_reg = Write multiple registers(0x10); Visibility = No}
    PANhoursOfWorkOsmos2 AT %QW9.2.50.0 [WordOutput] {ChannellName = Enter name}
  Register output module [ID2004] node 51, in %IB9.2.51 out %QB9.2.51 {ChannellName = Register; ModbusAddress = 328; Command_write_one_reg = Write multiple registers(0x10); Visibility = No}
    PANminutesOfWorkOsmos2 AT %QW9.2.51.0 [WordOutput] {ChannellName = Enter name}
  Register output module [ID2004] node 52, in %IB9.2.52 out %QB9.2.52 {ChannellName = Register; ModbusAddress = 329; Command_write_one_reg = Write multiple registers(0x10); Visibility = No}
    PANsecondsOfWorkOsmos2 AT %QW9.2.52.0 [WordOutput] {ChannellName = Enter name}
  Register output module [ID2004] node 53, in %IB9.2.53 out %QB9.2.53 {ChannellName = Register; ModbusAddress = 330; Command_write_one_reg = Write multiple registers(0x10); Visibility = No}
    PANtoNextStartOsmos2timer AT %QW9.2.53.0 [WordOutput] {ChannellName = Enter name}
  Register output module [ID2004] node 54, in %IB9.2.54 out %QB9.2.54 {ChannellName = Register; ModbusAddress = 331; Command_write_one_reg = Write multiple registers(0x10); Visibility = No}
    PANmainViewBools AT %QW9.2.54.0 [WordOutput] {ChannellName = Enter name}
  Real output module [ID2008] node 55, in %IB9.2.55 out %QB9.2.55 {ChannellName = float output module; ModbusAddress = 332; Command_write_regs = Preset multiple Registers (0x10); Visibility = No}
    PAN_BMT_Flow AT %QD9.2.55.0 [FloatOutput] {ChannellName = Enter name}
  32bit output module [ID2006] node 56, in %IB9.2.56 out %QB9.2.56 {ChannellName = 32 bit output module; ModbusAddress = 336; Command_write_regs = Preset multiple Registers (0x10); Visibility = No}
    PANalarms AT %QD9.2.56.0 [DWordOutput] {ChannellName = Enter name}
  Real output module [ID2008] node 57, in %IB9.2.57 out %QB9.2.57 {ChannellName = float output module; ModbusAddress = 338; Command_write_regs = Preset multiple Registers (0x10); Visibility = No}
    PAN_currentValue_PT0301startValue AT %QD9.2.57.0 [FloatOutput] {ChannellName = Enter name}
  Real output module [ID2008] node 58, in %IB9.2.58 out %QB9.2.58 {ChannellName = float output module; ModbusAddress = 340; Command_write_regs = Preset multiple Registers (0x10); Visibility = No}
    PAN_currentValue_FIT0303setValue AT %QD9.2.58.0 [FloatOutput] {ChannellName = Enter name}
  Real output module [ID2008] node 59, in %IB9.2.59 out %QB9.2.59 {ChannellName = float output module; ModbusAddress = 342; Command_write_regs = Preset multiple Registers (0x10); Visibility = No}
    PAN_currentValue_PT0302setMaxValue AT %QD9.2.59.0 [FloatOutput] {ChannellName = Enter name}
  Real output module [ID2008] node 60, in %IB9.2.60 out %QB9.2.60 {ChannellName = float output module; ModbusAddress = 344; Command_write_regs = Preset multiple Registers (0x10); Visibility = No}
    PAN_currentValue_PT0303setMaxValue AT %QD9.2.60.0 [FloatOutput] {ChannellName = Enter name}
  Real output module [ID2008] node 61, in %IB9.2.61 out %QB9.2.61 {ChannellName = float output module; ModbusAddress = 346; Command_write_regs = Preset multiple Registers (0x10); Visibility = No}
    PAN_currentValue_PT0304setMaxValue AT %QD9.2.61.0 [FloatOutput] {ChannellName = Enter name}
  Real output module [ID2008] node 62, in %IB9.2.62 out %QB9.2.62 {ChannellName = float output module; ModbusAddress = 348; Command_write_regs = Preset multiple Registers (0x10); Visibility = No}
    PAN_currentValue_FIT0303_SetCascade AT %QD9.2.62.0 [FloatOutput] {ChannellName = Enter name}
  Real output module [ID2008] node 63, in %IB9.2.63 out %QB9.2.63 {ChannellName = float output module; ModbusAddress = 350; Command_write_regs = Preset multiple Registers (0x10); Visibility = No}
    PAN_currentValue_KP_F_P030601 AT %QD9.2.63.0 [FloatOutput] {ChannellName = Enter name}
  Real output module [ID2008] node 64, in %IB9.2.64 out %QB9.2.64 {ChannellName = float output module; ModbusAddress = 352; Command_write_regs = Preset multiple Registers (0x10); Visibility = No}
    PAN_currentValue_I_F_P030601 AT %QD9.2.64.0 [FloatOutput] {ChannellName = Enter name}
  Real output module [ID2008] node 65, in %IB9.2.65 out %QB9.2.65 {ChannellName = float output module; ModbusAddress = 354; Command_write_regs = Preset multiple Registers (0x10); Visibility = No}
    PAN_currentValue_D_F_P030601 AT %QD9.2.65.0 [FloatOutput] {ChannellName = Enter name}
  Real output module [ID2008] node 66, in %IB9.2.66 out %QB9.2.66 {ChannellName = float output module; ModbusAddress = 356; Command_write_regs = Preset multiple Registers (0x10); Visibility = No}
    PAN_currentValue_KP_P_P030601 AT %QD9.2.66.0 [FloatOutput] {ChannellName = Enter name}
  Real output module [ID2008] node 67, in %IB9.2.67 out %QB9.2.67 {ChannellName = float output module; ModbusAddress = 358; Command_write_regs = Preset multiple Registers (0x10); Visibility = No}
    PAN_currentValue_I_P_P030601 AT %QD9.2.67.0 [FloatOutput] {ChannellName = Enter name}
  Real output module [ID2008] node 68, in %IB9.2.68 out %QB9.2.68 {ChannellName = float output module; ModbusAddress = 360; Command_write_regs = Preset multiple Registers (0x10); Visibility = No}
    PAN_currentValue_D_P_P030601 AT %QD9.2.68.0 [FloatOutput] {ChannellName = Enter name}
  Real output module [ID2008] node 69, in %IB9.2.69 out %QB9.2.69 {ChannellName = float output module; ModbusAddress = 362; Command_write_regs = Preset multiple Registers (0x10); Visibility = No}
    PAN_currentValue_KP_F_P030602 AT %QD9.2.69.0 [FloatOutput] {ChannellName = Enter name}
  Real output module [ID2008] node 70, in %IB9.2.70 out %QB9.2.70 {ChannellName = float output module; ModbusAddress = 364; Command_write_regs = Preset multiple Registers (0x10); Visibility = No}
    PAN_currentValue_I_F_P030602 AT %QD9.2.70.0 [FloatOutput] {ChannellName = Enter name}
  Real output module [ID2008] node 71, in %IB9.2.71 out %QB9.2.71 {ChannellName = float output module; ModbusAddress = 366; Command_write_regs = Preset multiple Registers (0x10); Visibility = No}
    PAN_currentValue_D_F_P030602 AT %QD9.2.71.0 [FloatOutput] {ChannellName = Enter name}
  Real output module [ID2008] node 72, in %IB9.2.72 out %QB9.2.72 {ChannellName = float output module; ModbusAddress = 368; Command_write_regs = Preset multiple Registers (0x10); Visibility = No}
    PAN_currentValue_KP_P_P030602 AT %QD9.2.72.0 [FloatOutput] {ChannellName = Enter name}
  Real output module [ID2008] node 73, in %IB9.2.73 out %QB9.2.73 {ChannellName = float output module; ModbusAddress = 370; Command_write_regs = Preset multiple Registers (0x10); Visibility = No}
    PAN_currentValue_I_P_P030602 AT %QD9.2.73.0 [FloatOutput] {ChannellName = Enter name}
  Real output module [ID2008] node 74, in %IB9.2.74 out %QB9.2.74 {ChannellName = float output module; ModbusAddress = 372; Command_write_regs = Preset multiple Registers (0x10); Visibility = No}
    PAN_currentValue_D_P_P030602 AT %QD9.2.74.0 [FloatOutput] {ChannellName = Enter name}
  Real output module [ID2008] node 75, in %IB9.2.75 out %QB9.2.75 {ChannellName = float output module; ModbusAddress = 374; Command_write_regs = Preset multiple Registers (0x10); Visibility = No}
    PAN_currentValue_setMaxPumpDosingValueP0302 AT %QD9.2.75.0 [FloatOutput] {ChannellName = Enter name}
  Real output module [ID2008] node 76, in %IB9.2.76 out %QB9.2.76 {ChannellName = float output module; ModbusAddress = 376; Command_write_regs = Preset multiple Registers (0x10); Visibility = No}
    PAN_currentValue_setKoeffProportionalityP0302 AT %QD9.2.76.0 [FloatOutput] {ChannellName = Enter name}
  Register output module [ID2004] node 77, in %IB9.2.77 out %QB9.2.77 {ChannellName = Register; ModbusAddress = 378; Command_write_one_reg = Write multiple registers(0x10); Visibility = No}
    PAN_currentValue_CHECKING_DELAY_TIME AT %QW9.2.77.0 [WordOutput] {ChannellName = Enter name}
  Register output module [ID2004] node 78, in %IB9.2.78 out %QB9.2.78 {ChannellName = Register; ModbusAddress = 379; Command_write_one_reg = Write multiple registers(0x10); Visibility = No}
    PAN_currentValue_DELAY_REPEATED_START_SEC AT %QW9.2.78.0 [WordOutput] {ChannellName = Enter name}
  Register output module [ID2004] node 79, in %IB9.2.79 out %QB9.2.79 {ChannellName = Register; ModbusAddress = 380; Command_write_one_reg = Write multiple registers(0x10); Visibility = No}
    PAN_currentValue_DELAY_TO_OFF_VALVE AT %QW9.2.79.0 [WordOutput] {ChannellName = Enter name}
  Register output module [ID2004] node 80, in %IB9.2.80 out %QB9.2.80 {ChannellName = Register; ModbusAddress = 381; Command_write_one_reg = Write multiple registers(0x10); Visibility = No}
    PAN_currentValue_DELAY_TO_CHECK_PT0301 AT %QW9.2.80.0 [WordOutput] {ChannellName = Enter name}
  Register output module [ID2004] node 81, in %IB9.2.81 out %QB9.2.81 {ChannellName = Register; ModbusAddress = 382; Command_write_one_reg = Write multiple registers(0x10); Visibility = No}
    PAN_currentValue_DELAY_TO_SWITCH_VALVE AT %QW9.2.81.0 [WordOutput] {ChannellName = Enter name}
  Register output module [ID2004] node 82, in %IB9.2.82 out %QB9.2.82 {ChannellName = Register; ModbusAddress = 383; Command_write_one_reg = Write multiple registers(0x10); Visibility = No}
    PAN_currentValue_DELAY_TO_CLOSE_VALVE AT %QW9.2.82.0 [WordOutput] {ChannellName = Enter name}
PAN_currentValue_FIT0301maxValue AT %QD9.2.83.0 [FloatOutput] {ChannellName = Enter name}
PAN_currentValue_FIT030201maxValue AT %QD9.2.84.0 [FloatOutput] {ChannellName = Enter name}
PAN_currentValue_FIT030301maxValue AT %QD9.2.85.0 [FloatOutput] {ChannellName = Enter name}
PAN_currentValue_FIT030202maxValue AT %QD9.2.86.0 [FloatOutput] {ChannellName = Enter name}
PAN_currentValue_FIT030302maxValue AT %QD9.2.87.0 [FloatOutput] {ChannellName = Enter name}
PAN_currentValue_QIT030101maxValue AT %QD9.2.88.0 [FloatOutput] {ChannellName = Enter name}
PAN_currentValue_QIT030102maxValue AT %QD9.2.89.0 [FloatOutput] {ChannellName = Enter name}
PAN_currentValue_PT030101maxValue AT %QD9.2.90.0 [FloatOutput] {ChannellName = Enter name}
PAN_currentValue_PT030201maxValue AT %QD9.2.91.0 [FloatOutput] {ChannellName = Enter name}
PAN_currentValue_PT030301maxValue AT %QD9.2.92.0 [FloatOutput] {ChannellName = Enter name}
PAN_currentValue_PT030401maxValue AT %QD9.2.93.0 [FloatOutput] {ChannellName = Enter name}
PAN_currentValue_PT030102maxValue AT %QD9.2.94.0 [FloatOutput] {ChannellName = Enter name}
PAN_currentValue_PT030202maxValue AT %QD9.2.95.0 [FloatOutput] {ChannellName = Enter name}
PAN_currentValue_PT030302maxValue AT %QD9.2.96.0 [FloatOutput] {ChannellName = Enter name}
PAN_currentValue_PT030402maxValue AT %QD9.2.97.0 [FloatOutput] {ChannellName = Enter name}
TCP [TCP_ID221] node 0, in %IB10.0.0 out %QB10.0.0 {ChannellName = TCP; RemotePort = 502; Visibility = No}
Float [Float] node 1, in %IB10.1 out %QB10.1 {ChannellName = float}
  ASU_FlowFromBMT AT %QD10.1.0 [FloatOutput] {ChannellName = Enter name}
4 byte [FourBytes] node 2, in %IB10.2 out %QB10.2 {ChannellName = 4 byte}
  ASU_alarms_from_ASU3_OPAN2 AT %QD10.2.0 [DWordOutput] {ChannellName = Enter name}
2 byte [Register] node 3, in %IB10.3 out %QB10.3 {ChannellName = 2 byte}
  ASU_Levels AT %QW10.3.0 [WordOutput] {ChannellName = Enter name}
2 byte [Register] node 4, in %IB10.4 out %QB10.4 {ChannellName = 2 byte}
  ASU_activators_OPAN2 AT %QW10.4.0 [WordOutput] {ChannellName = Enter name}
Float [Float] node 5, in %IB10.5 out %QB10.5 {ChannellName = float}
  ASU_FIT0301_OPAN2 AT %QD10.5.0 [FloatOutput] 6 ASU_FIT0301_ OPAN2 {ChannellName = Enter name}
Float [Float] node 6, in %IB10.6 out %QB10.6 {ChannellName = float}
  ASU_FIT030301_OPAN2 AT %QD10.6.0 [FloatOutput] {ChannellName = Enter name}
Float [Float] node 7, in %IB10.7 out %QB10.7 {ChannellName = float}
  ASU_FIT030302_OPAN2 AT %QD10.7.0 [FloatOutput] {ChannellName = Enter name}
Float [Float] node 8, in %IB10.8 out %QB10.8 {ChannellName = float}
  ASU_PT030101_OPAN2 AT %QD10.8.0 [FloatOutput] {ChannellName = Enter name}
Float [Float] node 9, in %IB10.9 out %QB10.9 {ChannellName = float}
  ASU_PT030201_OPAN2 AT %QD10.9.0 [FloatOutput] {ChannellName = Enter name}
Float [Float] node 10, in %IB10.10 out %QB10.10 {ChannellName = float}
  ASU_PT030301_OPAN2 AT %QD10.10.0 [FloatOutput] {ChannellName = Enter name}
Float [Float] node 11, in %IB10.11 out %QB10.11 {ChannellName = float}
  ASU_PT030102_OPAN2 AT %QD10.11.0 [FloatOutput] {ChannellName = Enter name}
Float [Float] node 12, in %IB10.12 out %QB10.12 {ChannellName = float}
  ASU_PT030202_OPAN2 AT %QD10.12.0 [FloatOutput] {ChannellName = Enter name}
Float [Float] node 13, in %IB10.13 out %QB10.13 {ChannellName = float}
  ASU_PT030302_OPAN2 AT %QD10.13.0 [FloatOutput] {ChannellName = Enter name}
Float [Float] node 14, in %IB10.14 out %QB10.14 {ChannellName = float}
  ASU_PT030401_OPAN2 AT %QD10.14.0 [FloatOutput] {ChannellName = Enter name}
Float [Float] node 15, in %IB10.15 out %QB10.15 {ChannellName = float}
  ASU_FIT030201_OPAN2 AT %QD10.15.0 [FloatOutput] {ChannellName = Enter name}
Float [Float] node 16, in %IB10.16 out %QB10.16 {ChannellName = float}
  ASU_QIT030101_OPAN2 AT %QD10.16.0 [FloatOutput] {ChannellName = Enter name}
Float [Float] node 17, in %IB10.17 out %QB10.17 {ChannellName = float}
  ASU_PT030402_OPAN2 AT %QD10.17.0 [FloatOutput] {ChannellName = Enter name}
Float [Float] node 18, in %IB10.18 out %QB10.18 {ChannellName = float}
  ASU_FIT030202_OPAN2 AT %QD10.18.0 [FloatOutput] {ChannellName = Enter name}
Float [Float] node 19, in %IB10.19 out %QB10.19 {ChannellName = float}
  ASU_QIT030102_OPAN2 AT %QD10.19.0 [FloatOutput] {ChannellName = Enter name}
4 byte [FourBytes] node 20, in %IB10.20 out %QB10.20 {ChannellName = 4 byte}
  ASU_mainPageStatusWord_OPAN2 AT %QD10.20.0 [DWordOutput] {ChannellName = Enter name}
Float [Float] node 21, in %IB10.21 out %QB10.21 {ChannellName = float}
  ASU_counterP030101_OPAN2 AT %QD10.21.0 [FloatOutput] {ChannellName = Enter name}
Float [Float] node 22, in %IB10.22 out %QB10.22 {ChannellName = float}
  ASU_counterP030102_OPAN2 AT %QD10.22.0 [FloatOutput] {ChannellName = Enter name}
2 byte [Register] node 23, in %IB10.23 out %QB10.23 {ChannellName = 2 byte}
  ASU_daysOfWorkP030101_OPAN2 AT %QW10.23.0 [WordOutput] {ChannellName = Enter name}
2 byte [Register] node 24, in %IB10.24 out %QB10.24 {ChannellName = 2 byte}
  ASU_hoursOfWorkP030101_OPAN2 AT %QW10.24.0 [WordOutput] {ChannellName = Enter name}
2 byte [Register] node 25, in %IB10.25 out %QB10.25 {ChannellName = 2 byte}
  ASU_minutesOfWorkP030101_OPAN2 AT %QW10.25.0 [WordOutput] {ChannellName = Enter name}
2 byte [Register] node 26, in %IB10.26 out %QB10.26 {ChannellName = 2 byte}
  ASU_secondsOfWorkP030101_OPAN2 AT %QW10.26.0 [WordOutput] {ChannellName = Enter name}
2 byte [Register] node 27, in %IB10.27 out %QB10.27 {ChannellName = 2 byte}
  ASU_toNextStartP030101timer_OPAN2 AT %QW10.27.0 [WordOutput] {ChannellName = Enter name}
2 byte [Register] node 28, in %IB10.28 out %QB10.28 {ChannellName = 2 byte}
  ASU_daysOfWorkP030102_OPAN2 AT %QW10.28.0 [WordOutput] {ChannellName = Enter name}
2 byte [Register] node 29, in %IB10.29 out %QB10.29 {ChannellName = 2 byte}
  ASU_hoursOfWorkP030102_OPAN2 AT %QW10.29.0 [WordOutput] {ChannellName = Enter name}
2 byte [Register] node 30, in %IB10.30 out %QB10.30 {ChannellName = 2 byte}
  ASU_minutesOfWorkP030102_OPAN2 AT %QW10.30.0 [WordOutput] {ChannellName = Enter name}
2 byte [Register] node 31, in %IB10.31 out %QB10.31 {ChannellName = 2 byte}
  ASU_secondsOfWorkP030102_OPAN2 AT %QW10.31.0 [WordOutput] {ChannellName = Enter name}
2 byte [Register] node 32, in %IB10.32 out %QB10.32 {ChannellName = 2 byte}
  ASU_toNextStartP030102timer_OPAN2 AT %QW10.32.0 [WordOutput] {ChannellName = Enter name}
2 byte [Register] node 33, in %IB10.33 out %QB10.33 {ChannellName = 2 byte}
  ASU_statWordP0301_OPAN2 AT %QW10.33.0 [WordOutput] {ChannellName = Enter name}
2 byte [Register] node 34, in %IB10.34 out %QB10.34 {ChannellName = 2 byte}
  ASU_setWordP0301_OPAN2 AT %QW10.34.0 [WordOutput] {ChannellName = Enter name}
Float [Float] node 35, in %IB10.35 out %QB10.35 {ChannellName = float}
  ASU_counterP030201_OPAN2 AT %QD10.35.0 [FloatOutput] {ChannellName = Enter name}
Float [Float] node 36, in %IB10.36 out %QB10.36 {ChannellName = float}
  ASU_counterP030202_OPAN2 AT %QD10.36.0 [FloatOutput] {ChannellName = Enter name}
2 byte [Register] node 37, in %IB10.37 out %QB10.37 {ChannellName = 2 byte}
  ASU_daysOfWorkP030201_OPAN2 AT %QW10.37.0 [WordOutput] {ChannellName = Enter name}
2 byte [Register] node 38, in %IB10.38 out %QB10.38 {ChannellName = 2 byte}
  ASU_hoursOfWorkP030201_OPAN2 AT %QW10.38.0 [WordOutput] {ChannellName = Enter name}
2 byte [Register] node 39, in %IB10.39 out %QB10.39 {ChannellName = 2 byte}
  ASU_minutesOfWorkP030201_OPAN2 AT %QW10.39.0 [WordOutput] {ChannellName = Enter name}
2 byte [Register] node 40, in %IB10.40 out %QB10.40 {ChannellName = 2 byte}
  ASU_secondsOfWorkP030201_OPAN2 AT %QW10.40.0 [WordOutput] {ChannellName = Enter name}
2 byte [Register] node 41, in %IB10.41 out %QB10.41 {ChannellName = 2 byte}
  ASU_toNextStartP030201timer_OPAN2 AT %QW10.41.0 [WordOutput] {ChannellName = Enter name}
2 byte [Register] node 42, in %IB10.42 out %QB10.42 {ChannellName = 2 byte}
  ASU_daysOfWorkP030202_OPAN2 AT %QW10.42.0 [WordOutput] {ChannellName = Enter name}
2 byte [Register] node 43, in %IB10.43 out %QB10.43 {ChannellName = 2 byte}
  ASU_hoursOfWorkP030202_OPAN2 AT %QW10.43.0 [WordOutput] {ChannellName = Enter name}
2 byte [Register] node 44, in %IB10.44 out %QB10.44 {ChannellName = 2 byte}
  ASU_minutesOfWorkP030202_OPAN2 AT %QW10.44.0 [WordOutput] {ChannellName = Enter name}
2 byte [Register] node 45, in %IB10.45 out %QB10.45 {ChannellName = 2 byte}
  ASU_secondsOfWorkP030202_OPAN2 AT %QW10.45.0 [WordOutput] {ChannellName = Enter name}
2 byte [Register] node 46, in %IB10.46 out %QB10.46 {ChannellName = 2 byte}
  ASU_toNextStartP030202timer_OPAN2 AT %QW10.46.0 [WordOutput] {ChannellName = Enter name}
2 byte [Register] node 47, in %IB10.47 out %QB10.47 {ChannellName = 2 byte}
  ASU_statWordP0302_OPAN2 AT %QW10.47.0 [WordOutput] {ChannellName = Enter name}
2 byte [Register] node 48, in %IB10.48 out %QB10.48 {ChannellName = 2 byte}
  AT %QW10.48.0 [WordOutput] {ChannellName = Enter name}
Float [Float] node 49, in %IB10.49 out %QB10.49 {ChannellName = float}
  ASU_currentValue_setMaxPumpDosingValueP0302_OPAN2 AT %QD10.49.0 [FloatOutput] {ChannellName = Enter name}
Float [Float] node 50, in %IB10.50 out %QB10.50 {ChannellName = float}
  ASU_currentValue_setKoeffProportionalityP0302_OPAN2 AT %QD10.50.0 [FloatOutput] {ChannellName = Enter name}
Float [Float] node 51, in %IB10.51 out %QB10.51 {ChannellName = float}
  ASU_setMaxPumpDosingValueP0302_OPAN2 AT %QD10.51.0 [FloatOutput] {ChannellName = Enter name}
Float [Float] node 52, in %IB10.52 out %QB10.52 {ChannellName = float}
  ASU_setKoeffProportionalityP0302_OPAN2 AT %QD10.52.0 [FloatOutput] {ChannellName = Enter name}
2 byte [Register] node 53, in %IB10.53 out %QB10.53 {ChannellName = 2 byte}
  ASU_setWordP0302_OPAN2 AT %QW10.53.0 [WordOutput] {ChannellName = Enter name}
2 byte [Register] node 54, in %IB10.54 out %QB10.54 {ChannellName = 2 byte}
  ASU_currentValue_CHECKING_DELAY_TIME_OPAN2 AT %QW10.54.0 [WordOutput] {ChannellName = Enter name}
2 byte [Register] node 55, in %IB10.55 out %QB10.55 {ChannellName = 2 byte}
  ASU_currentValue_DELAY_REPEATED_START_SEC_OPAN2 AT %QW10.55.0 [WordOutput] {ChannellName = Enter name}
2 byte [Register] node 56, in %IB10.56 out %QB10.56 {ChannellName = 2 byte}
  ASU_currentValue_DELAY_TO_OFF_VALVE_OPAN2 AT %QW10.56.0 [WordOutput] {ChannellName = Enter name}
2 byte [Register] node 57, in %IB10.57 out %QB10.57 {ChannellName = 2 byte}
  ASU_currentValue_DELAY_TO_CHECK_PT0301_OPAN2 AT %QW10.57.0 [WordOutput] {ChannellName = Enter name}
2 byte [Register] node 58, in %IB10.58 out %QB10.58 {ChannellName = 2 byte}
  ASU_currentValue_DELAY_TO_SWITCH_VALVE_OPAN2 AT %QW10.58.0 [WordOutput] {ChannellName = Enter name}
2 byte [Register] node 59, in %IB10.59 out %QB10.59 {ChannellName = 2 byte}
  ASU_currentValue_DELAY_TO_CLOSE_VALVE_OPAN2 AT %QW10.59.0 [WordOutput] {ChannellName = Enter name}
2 byte [Register] node 60, in %IB10.60 out %QB10.60 {ChannellName = 2 byte}
  ASU_CHECKING_DELAY_TIME_OPAN2 AT %QW10.60.0 [WordOutput] {ChannellName = Enter name}
2 byte [Register] node 61, in %IB10.61 out %QB10.61 {ChannellName = 2 byte}
  ASU_DELAY_REPEATED_START_SEC_OPAN2 AT %QW10.61.0 [WordOutput] {ChannellName = Enter name}
2 byte [Register] node 62, in %IB10.62 out %QB10.62 {ChannellName = 2 byte}
  ASU_DELAY_TO_OFF_VALVE_OPAN2 AT %QW10.62.0 [WordOutput] {ChannellName = Enter name}
2 byte [Register] node 63, in %IB10.63 out %QB10.63 {ChannellName = 2 byte}
  ASU_DELAY_TO_CHECK_PT0301_OPAN2 AT %QW10.63.0 [WordOutput] {ChannellName = Enter name}
2 byte [Register] node 64, in %IB10.64 out %QB10.64 {ChannellName = 2 byte}
  ASU_DELAY_TO_SWITCH_VALVE_OPAN2 AT %QW10.64.0 [WordOutput] {ChannellName = Enter name}
2 byte [Register] node 65, in %IB10.65 out %QB10.65 {ChannellName = 2 byte}
  ASU_DELAY_TO_CLOSE_VALVE_OPAN2 AT %QW10.65.0 [WordOutput] {ChannellName = Enter name}
2 byte [Register] node 66, in %IB10.66 out %QB10.66 {ChannellName = 2 byte}
  AT %QW10.66.0 [WordOutput] {ChannellName = Enter name}
Float [Float] node 67, in %IB10.67 out %QB10.67 {ChannellName = float}
  ASU_currentValue_FIT0301maxValue_OPAN2 AT %QD10.67.0 [FloatOutput] {ChannellName = Enter name}
Float [Float] node 68, in %IB10.68 out %QB10.68 {ChannellName = float}
  ASU_currentValue_FIT030201maxValue_OPAN2 AT %QD10.68.0 [FloatOutput] {ChannellName = Enter name}
Float [Float] node 69, in %IB10.69 out %QB10.69 {ChannellName = float}
  ASU_currentValue_FIT030301maxValue_OPAN2 AT %QD10.69.0 [FloatOutput] {ChannellName = Enter name}
Float [Float] node 70, in %IB10.70 out %QB10.70 {ChannellName = float}
  ASU_currentValue_FIT030202maxValue_OPAN2 AT %QD10.70.0 [FloatOutput] {ChannellName = Enter name}
Float [Float] node 71, in %IB10.71 out %QB10.71 {ChannellName = float}
  ASU_currentValue_FIT030302maxValue_OPAN2 AT %QD10.71.0 [FloatOutput] {ChannellName = Enter name}
Float [Float] node 72, in %IB10.72 out %QB10.72 {ChannellName = float}
  ASU_currentValue_QIT030101maxValue_OPAN2 AT %QD10.72.0 [FloatOutput] {ChannellName = Enter name}
Float [Float] node 73, in %IB10.73 out %QB10.73 {ChannellName = float}
  ASU_currentValue_QIT030102maxValue_OPAN2 AT %QD10.73.0 [FloatOutput] {ChannellName = Enter name}
Float [Float] node 74, in %IB10.74 out %QB10.74 {ChannellName = float}
  ASU_currentValue_PT030101maxValue_OPAN2 AT %QD10.74.0 [FloatOutput] {ChannellName = Enter name}
Float [Float] node 75, in %IB10.75 out %QB10.75 {ChannellName = float}
  ASU_currentValue_PT030201maxValue_OPAN2 AT %QD10.75.0 [FloatOutput] {ChannellName = Enter name}
Float [Float] node 76, in %IB10.76 out %QB10.76 {ChannellName = float}
  ASU_currentValue_PT030301maxValue_OPAN2 AT %QD10.76.0 [FloatOutput] {ChannellName = Enter name}
Float [Float] node 77, in %IB10.77 out %QB10.77 {ChannellName = float}
  ASU_currentValue_PT030401maxValue_OPAN2 AT %QD10.77.0 [FloatOutput] {ChannellName = Enter name}
Float [Float] node 78, in %IB10.78 out %QB10.78 {ChannellName = float}
  ASU_currentValue_PT030102maxValue_OPAN2 AT %QD10.78.0 [FloatOutput] {ChannellName = Enter name}
Float [Float] node 79, in %IB10.79 out %QB10.79 {ChannellName = float}
  ASU_currentValue_PT030202maxValue_OPAN2 AT %QD10.79.0 [FloatOutput] {ChannellName = Enter name}
Float [Float] node 80, in %IB10.80 out %QB10.80 {ChannellName = float}
  ASU_currentValue_PT030302maxValue_OPAN2 AT %QD10.80.0 [FloatOutput] {ChannellName = Enter name}
Float [Float] node 81, in %IB10.81 out %QB10.81 {ChannellName = float}
  ASU_currentValue_PT030402maxValue_OPAN2 AT %QD10.81.0 [FloatOutput] {ChannellName = Enter name}
Float [Float] node 82, in %IB10.82 out %QB10.82 {ChannellName = float}
  ASU_set_FIT0301maxValue_OPAN2 AT %QD10.82.0 [FloatOutput] {ChannellName = Enter name}
Float [Float] node 83, in %IB10.83 out %QB10.83 {ChannellName = float}
  ASU_set_FIT030201maxValue_OPAN2 AT %QD10.83.0 [FloatOutput] {ChannellName = Enter name}
Float [Float] node 84, in %IB10.84 out %QB10.84 {ChannellName = float}
  ASU_set_FIT030301maxValue_OPAN2 AT %QD10.84.0 [FloatOutput] {ChannellName = Enter name}
Float [Float] node 85, in %IB10.85 out %QB10.85 {ChannellName = float}
  ASU_set_FIT030202maxValue_OPAN2 AT %QD10.85.0 [FloatOutput] {ChannellName = Enter name}
Float [Float] node 86, in %IB10.86 out %QB10.86 {ChannellName = float}
  ASU_set_FIT030302maxValue_OPAN2 AT %QD10.86.0 [FloatOutput] {ChannellName = Enter name}
Float [Float] node 87, in %IB10.87 out %QB10.87 {ChannellName = float}
  ASU_set_QIT030101maxValue_OPAN2 AT %QD10.87.0 [FloatOutput] {ChannellName = Enter name}
Float [Float] node 88, in %IB10.88 out %QB10.88 {ChannellName = float}
  ASU_set_QIT030102maxValue_OPAN2 AT %QD10.88.0 [FloatOutput] {ChannellName = Enter name}
Float [Float] node 89, in %IB10.89 out %QB10.89 {ChannellName = float}
  ASU_set_PT030101maxValue_OPAN2 AT %QD10.89.0 [FloatOutput] {ChannellName = Enter name}
Float [Float] node 90, in %IB10.90 out %QB10.90 {ChannellName = float}
  ASU_set_PT030201maxValue_OPAN2 AT %QD10.90.0 [FloatOutput] {ChannellName = Enter name}
Float [Float] node 91, in %IB10.91 out %QB10.91 {ChannellName = float}
  ASU_set_PT030301maxValue_OPAN2 AT %QD10.91.0 [FloatOutput] {ChannellName = Enter name}
Float [Float] node 92, in %IB10.92 out %QB10.92 {ChannellName = float}
  ASU_set_PT030401maxValue_OPAN2 AT %QD10.92.0 [FloatOutput] {ChannellName = Enter name}
Float [Float] node 93, in %IB10.93 out %QB10.93 {ChannellName = float}
  ASU_set_PT030102maxValue_OPAN2 AT %QD10.93.0 [FloatOutput] {ChannellName = Enter name}
Float [Float] node 94, in %IB10.94 out %QB10.94 {ChannellName = float}
  ASU_set_PT030202maxValue_OPAN2 AT %QD10.94.0 [FloatOutput] {ChannellName = Enter name}
Float [Float] node 95, in %IB10.95 out %QB10.95 {ChannellName = float}
  ASU_set_PT030302maxValue_OPAN2 AT %QD10.95.0 [FloatOutput] {ChannellName = Enter name}
Float [Float] node 96, in %IB10.96 out %QB10.96 {ChannellName = float}
  ASU_set_PT030402maxValue_OPAN2 AT %QD10.96.0 [FloatOutput] {ChannellName = Enter name}
Float [Float] node 97, in %IB10.97 out %QB10.97 {ChannellName = float}
  ASU_counterPV030701_OPAN2 AT %QD10.97.0 [FloatOutput] {ChannellName = Enter name}
Float [Float] node 98, in %IB10.98 out %QB10.98 {ChannellName = float}
  ASU_counterPV030702_OPAN2 AT %QD10.98.0 [FloatOutput] {ChannellName = Enter name}
2 byte [Register] node 99, in %IB10.99 out %QB10.99 {ChannellName = 2 byte}
  ASU_statWordPV0307_OPAN2 AT %QW10.99.0 [WordOutput] {ChannellName = Enter name}
2 byte [Register] node 100, in %IB10.100 out %QB10.100 {ChannellName = 2 byte}
  ASU_daysOfWorkPV030701_OPAN2 AT %QW10.100.0 [WordOutput] {ChannellName = Enter name}
2 byte [Register] node 101, in %IB10.101 out %QB10.101 {ChannellName = 2 byte}
  ASU_hoursOfWorkPV030701_OPAN2 AT %QW10.101.0 [WordOutput] {ChannellName = Enter name}
2 byte [Register] node 102, in %IB10.102 out %QB10.102 {ChannellName = 2 byte}
  ASU_minutesOfWorkPV030701_OPAN2 AT %QW10.102.0 [WordOutput] {ChannellName = Enter name}
2 byte [Register] node 103, in %IB10.103 out %QB10.103 {ChannellName = 2 byte}
  ASU_secondsOfWorkPV030701_OPAN2 AT %QW10.103.0 [WordOutput] {ChannellName = Enter name}
2 byte [Register] node 104, in %IB10.104 out %QB10.104 {ChannellName = 2 byte}
  ASU_toNextStartPV030701timer_OPAN2 AT %QW10.104.0 [WordOutput] {ChannellName = Enter name}
2 byte [Register] node 105, in %IB10.105 out %QB10.105 {ChannellName = 2 byte}
  ASU_daysOfWorkPV030702_OPAN2 AT %QW10.105.0 [WordOutput] {ChannellName = Enter name}
2 byte [Register] node 106, in %IB10.106 out %QB10.106 {ChannellName = 2 byte}
  ASU_hoursOfWorkPV030702_OPAN2 AT %QW10.106.0 [WordOutput] {ChannellName = Enter name}
2 byte [Register] node 107, in %IB10.107 out %QB10.107 {ChannellName = 2 byte}
  ASU_minutesOfWorkPV030702_OPAN2 AT %QW10.107.0 [WordOutput] {ChannellName = Enter name}
2 byte [Register] node 108, in %IB10.108 out %QB10.108 {ChannellName = 2 byte}
  ASU_secondsOfWorkPV030702_OPAN2 AT %QW10.108.0 [WordOutput] {ChannellName = Enter name}
2 byte [Register] node 109, in %IB10.109 out %QB10.109 {ChannellName = 2 byte}
  ASU_toNextStartPV030702timer_OPAN2 AT %QW10.109.0 [WordOutput] {ChannellName = Enter name}
2 byte [Register] node 110, in %IB10.110 out %QB10.110 {ChannellName = 2 byte}
  ASU_setWordPV0307_OPAN2 AT %QW10.110.0 [WordOutput] {ChannellName = Enter name}
Float [Float] node 111, in %IB10.111 out %QB10.111 {ChannellName = float}
  ASU_active_KP_F_P030601_OPAN2 AT %QD10.111.0 [FloatOutput] {ChannellName = Enter name}
Float [Float] node 112, in %IB10.112 out %QB10.112 {ChannellName = float}
  ASU_active_I_F_P030601_OPAN2 AT %QD10.112.0 [FloatOutput] {ChannellName = Enter name}
Float [Float] node 113, in %IB10.113 out %QB10.113 {ChannellName = float}
  ASU_active_D_F_P030601_OPAN2 AT %QD10.113.0 [FloatOutput] {ChannellName = Enter name}
Float [Float] node 114, in %IB10.114 out %QB10.114 {ChannellName = float}
  ASU_active_KP_P_P030601_OPAN2 AT %QD10.114.0 [FloatOutput] {ChannellName = Enter name}
Float [Float] node 115, in %IB10.115 out %QB10.115 {ChannellName = float}
  ASU_active_I_P_P030601_OPAN2 AT %QD10.115.0 [FloatOutput] {ChannellName = Enter name}
Float [Float] node 116, in %IB10.116 out %QB10.116 {ChannellName = float}
  ASU_active_D_P_P030601_OPAN2 AT %QD10.116.0 [FloatOutput] {ChannellName = Enter name}
Float [Float] node 117, in %IB10.117 out %QB10.117 {ChannellName = float}
  ASU_PAN_KP_F_P030601_OPAN2 AT %QD10.117.0 [FloatOutput] {ChannellName = Enter name}
Float [Float] node 118, in %IB10.118 out %QB10.118 {ChannellName = float}
  ASU_PAN_I_F_P030601_OPAN2 AT %QD10.118.0 [FloatOutput] {ChannellName = Enter name}
Float [Float] node 119, in %IB10.119 out %QB10.119 {ChannellName = float}
  ASU_PAN_D_F_P030601_OPAN2 AT %QD10.119.0 [FloatOutput] {ChannellName = Enter name}
Float [Float] node 120, in %IB10.120 out %QB10.120 {ChannellName = float}
  ASU_PAN_KP_P_P030601_OPAN2 AT %QD10.120.0 [FloatOutput] {ChannellName = Enter name}
Float [Float] node 121, in %IB10.121 out %QB10.121 {ChannellName = float}
  ASU_PAN_I_P_P030601_OPAN2 AT %QD10.121.0 [FloatOutput] {ChannellName = Enter name}
Float [Float] node 122, in %IB10.122 out %QB10.122 {ChannellName = float}
  ASU_PAN_D_P_P030601_OPAN2 AT %QD10.122.0 [FloatOutput] {ChannellName = Enter name}
Float [Float] node 123, in %IB10.123 out %QB10.123 {ChannellName = float}
  ASU_active_KP_F_P030602_OPAN2 AT %QD10.123.0 [FloatOutput] {ChannellName = Enter name}
Float [Float] node 124, in %IB10.124 out %QB10.124 {ChannellName = float}
  ASU_active_I_F_P030602_OPAN2 AT %QD10.124.0 [FloatOutput] {ChannellName = Enter name}
Float [Float] node 125, in %IB10.125 out %QB10.125 {ChannellName = float}
  ASU_active_D_F_P030602_OPAN2 AT %QD10.125.0 [FloatOutput] {ChannellName = Enter name}
Float [Float] node 126, in %IB10.126 out %QB10.126 {ChannellName = float}
  ASU_active_KP_P_P030602_OPAN2 AT %QD10.126.0 [FloatOutput] {ChannellName = Enter name}
Float [Float] node 127, in %IB10.127 out %QB10.127 {ChannellName = float}
  ASU_active_I_P_P030602_OPAN2 AT %QD10.127.0 [FloatOutput] {ChannellName = Enter name}
Float [Float] node 128, in %IB10.128 out %QB10.128 {ChannellName = float}
  ASU_active_D_P_P030602_OPAN2 AT %QD10.128.0 [FloatOutput] {ChannellName = Enter name}
Float [Float] node 129, in %IB10.129 out %QB10.129 {ChannellName = float}
  ASU_PAN_KP_F_P030602_OPAN2 AT %QD10.129.0 [FloatOutput] {ChannellName = Enter name}
Float [Float] node 130, in %IB10.130 out %QB10.130 {ChannellName = float}
  ASU_PAN_I_F_P030602_OPAN2 AT %QD10.130.0 [FloatOutput] {ChannellName = Enter name}
Float [Float] node 131, in %IB10.131 out %QB10.131 {ChannellName = float}
  ASU_PAN_D_F_P030602_OPAN2 AT %QD10.131.0 [FloatOutput] {ChannellName = Enter name}
Float [Float] node 132, in %IB10.132 out %QB10.132 {ChannellName = float}
  ASU_PAN_KP_P_P030602_OPAN2 AT %QD10.132.0 [FloatOutput] {ChannellName = Enter name}
Float [Float] node 133, in %IB10.133 out %QB10.133 {ChannellName = float}
  ASU_PAN_I_P_P030602_OPAN2 AT %QD10.133.0 [FloatOutput] {ChannellName = Enter name}
Float [Float] node 134, in %IB10.134 out %QB10.134 {ChannellName = float}
  ASU_PAN_D_P_P030602_OPAN2 AT %QD10.134.0 [FloatOutput] {ChannellName = Enter name}
Float [Float] node 135, in %IB10.135 out %QB10.135 {ChannellName = float}
  ASU_PAN_BMT_Flow_OPAN2 AT %QD10.135.0 [FloatOutput] {ChannellName = Enter name}
Float [Float] node 136, in %IB10.136 out %QB10.136 {ChannellName = float}
  ASU_currentValue_PT0301startValue_OPAN2 AT %QD10.136.0 [FloatOutput] {ChannellName = Enter name}
Float [Float] node 137, in %IB10.137 out %QB10.137 {ChannellName = float}
  ASU_currentValue_FIT0303setValue_OPAN2 AT %QD10.137.0 [FloatOutput] {ChannellName = Enter name}
Float [Float] node 138, in %IB10.138 out %QB10.138 {ChannellName = float}
  ASU_currentValue_PT0302setMaxValue_OPAN2 AT %QD10.138.0 [FloatOutput] {ChannellName = Enter name}
Float [Float] node 139, in %IB10.139 out %QB10.139 {ChannellName = float}
  ASU_currentValue_PT0303setMaxValue_OPAN2 AT %QD10.139.0 [FloatOutput] {ChannellName = Enter name}
Float [Float] node 140, in %IB10.140 out %QB10.140 {ChannellName = float}
  ASU_currentValue_PT0304setMaxValue_OPAN2 AT %QD10.140.0 [FloatOutput] {ChannellName = Enter name}
Float [Float] node 141, in %IB10.141 out %QB10.141 {ChannellName = float}
  ASU_currentValue_FIT0303_SetCascade_OPAN2 AT %QD10.141.0 [FloatOutput] {ChannellName = Enter name}
Float [Float] node 142, in %IB10.142 out %QB10.142 {ChannellName = float}
  ASU_PT0301startValue_OPAN2 AT %QD10.142.0 [FloatOutput] {ChannellName = Enter name}
Float [Float] node 143, in %IB10.143 out %QB10.143 {ChannellName = float}
  ASU_FIT0303setValue_OPAN2 AT %QD10.143.0 [FloatOutput] {ChannellName = Enter name}
Float [Float] node 144, in %IB10.144 out %QB10.144 {ChannellName = float}
  ASU_PT0302setValue_OPAN2 AT %QD10.144.0 [FloatOutput] {ChannellName = Enter name}
Float [Float] node 145, in %IB10.145 out %QB10.145 {ChannellName = float}
  ASU_PT0303setValue_OPAN2 AT %QD10.145.0 [FloatOutput] {ChannellName = Enter name}
Float [Float] node 146, in %IB10.146 out %QB10.146 {ChannellName = float}
  ASU_PT0304setValue_OPAN2 AT %QD10.146.0 [FloatOutput] {ChannellName = Enter name}
Float [Float] node 147, in %IB10.147 out %QB10.147 {ChannellName = float}
  ASU_FIT0303_SetCascade_OPAN2 AT %QD10.147.0 [FloatOutput] {ChannellName = Enter name}
*)

(* POU PLC_PRG, CFC *)
PROGRAM PLC_PRG
VAR
	P0301: RichTwoPumpManager;		(*управление насосами Р03.01 на входе в осмос*)
	resetAlarms: BOOL;		(*Сброс аварий в осмос 2 (МЕ03)*)
	delayCheckIfP030101works: TON;		(*задержка на разгон насоса Р03.01/01*)
	delayCheckIfP030102works: TON;		(*задержка на разгон насоса Р03.01/02*)
	lowLevelV0207: BOOL;		(*низкий уровень в емкости V02.07, сигнал из АСУ-2 осмос-1*)
	highLevelV0601: BOOL;		(*высокий уровень в емкости V06.01 сигнал из АСУ-1 общий.*)
	highLevelV0401: BOOL;		(*высокий уровень в емкости V04.01, сигнал из МЕ04, от БМТ.*)
	toNextStartP030101timer: WORD;		(*Обратный отсчет до возможности повторного пуска насоса Р03.01/01*)
	toNextStartP030102timer: WORD;		(*обратный отсчет до возможности повторного пуска насоса Р03.01/02*)
	FIT0301realValue: REAL;		(*Показания расходомера FIT03.01/01 на входе в осмос 2.
			Для управления производительностью НД Р03.02 (1 и 2).*)
	P0302: RichTwoPumpManager;		(*блок управления доз.насосами Р03.02/01 и Р03.02/02.*)
	P0302dos: DosingPumpProportional;		(*блок управления промзводительностью доз.насосов Р03.02.*)
	dosingErrorP0302: BOOL;		(*Ошибка производительности дозирования (неверно заданы значения производительности насоса,
производительность доз.насоса не соответствует расходу.*)
	initializer: R_TRIG;		(*триггер дающий импульс при включении программы.*)
	alarmP0302: BOOL;		(*авария обоих доз.насосов Р03..02 на входе в осмос*)
	osmosTotalAlarm: BOOL;		(*авария обоих осмосов*)
	controlAIpt030101: ControlAI;
	PT030101realValue: REAL;		(*Показания датчика РТ03.01/01, МПа (Бар)*)
	PT030101alarm: BOOL;		(*авария датчика РТ03.01/01*)
	controlAIpt030201: ControlAI;
	PT030201realValue: REAL;
	PT030201alarm: BOOL;
	controlAIpt030301: ControlAI;
	PT030301realValue: REAL;
	PT030301alarm: BOOL;
	controlAIpt030401: ControlAI;
	PT030401realValue: REAL;
	PT030401alarm: BOOL;
	controlAIqit030101: ControlAI;
	QIT030101realValue: REAL;
	QIT030101alarm: BOOL;
	controlAIfit030201: ControlAI;
	FIT030201realValue: REAL;
	FIT030201alarm: BOOL;
	controlAIfit030301: ControlAI;
	FIT030301realValue: REAL;
	FIT030301alarm: BOOL;
	osmos2sensorsAlarm: BOOL;		(*Авария датчиков осмос 2.
			в DD2 (ПР102) есть авария одного из датчиков.*)
	osmosManager: RichTwoPumpManager;
	toNextStartOsmos1timer: WORD;
	toNextStartOsmos2timer: WORD;
	minutesOfWorkOsmos2: WORD;
	secondsOfWorkOsmos2: WORD;
	osmos1SensorAlarm: BOOL;		(*Авария оборудования основного осмоса.*)
	osmos1EquipmentAlarm: BOOL;		(*Авария оборудования основного осмоса.*)
	osmos2EquipmentAlarm: BOOL;		(*авария оборудования резервного осмоса*)
	tofValve12: TOF;
	tonValve14: TON;
	tofValve14: TOF;
	tonValve18: TON;
	startP0302: BOOL;		(*сигнал на запуск насосов-дозаторов Р03.02*)
	tonPT030101: TON;
	lowPT030101_P030101: BOOL;		(*давление на РТ030101 не достигло значения для старта при
			активном насосе Р03.01/01*)
	lowPT030101_P030102: BOOL;		(*давление на РТ030101 не достигло значения для старта при
			активном насосе Р03.01/02*)
	tonSwitchValve1413: TON;
	valve1413switcher: IfBOOL;
	delayToSwitchValve14to13: TOF;
	F_P030601: PID;		(*PID регулятор по расходу Р03.06/01*)
	P_P030601: PID;		(*PID регулятор по давлению Р03.06/01*)
	Yout_F_P030601: REAL;		(*задание ПИД по расходу для Р030601*)
	Yout_P_P030601: REAL;		(*выход регулировки по давлению Р03.06/01, 0...100*)
	Yout_Total_P030601: REAL;		(*итоговый управляющий сигнал производительность Р03.06/01*)
	Yout_F_P030602: REAL;		(*задание ПИД по расходу для Р030602*)
	Yout_P_P030602: REAL;		(*выход регулировки по давлению Р03.06/02, 0...100*)
	Yout_Total_P030602: REAL;		(*итоговый управляющий сигнал производительность Р03.06/02*)
	P030601alarm: BOOL;		(*авария насоса Р03.06/01*)
	P030602alarm: BOOL;		(*авария насоса Р03.06/02*)
	P030601start: BOOL;		(*сигнал на запуск насоса Р03.06/01*)
	P030602start: BOOL;		(*сигнал на запуск насоса Р03.06/02*)
	osmos1AlarmPT030301: BOOL;		(*авария основного осмоса по макс давлению датчика РТ03.03/01*)
	osmos1AlarmPT030401: BOOL;		(*авария основного осмоса по макс давлению датчика РТ03.04/01*)
	osmos2AlarmPT030302: BOOL;		(*авария основного осмоса по макс давлению датчика РТ03.03/02*)
	osmos2AlarmPT030402: BOOL;		(*авария основного осмоса по макс давлению датчика РТ03.04/02*)
	tofValve18: TOF;
	HoldingToEndProcValve: TOF;
	tonValve17: TON;
	tonValve18rez: TON;
	tofValve18rez: TOF;
	tofValve17: TOF;
	tofValve15: TOF;
	lowPT030102_P030101: BOOL;		(*авария насоса Р03.01/01 по низкому давлению РТ03.01/02*)
	lowPT030102_P030102: BOOL;		(*авария насоса Р03.01/02 по низкому давлению РТ03.01/02*)
	PT030102realValue: REAL;		(*давление РТ03.01/02 из DD2*)
	tonSwitchValve1716: TON;
	HoldingToEndProcValveRez: TOF;
	tonPT030102: TON;
	valve1716switcher: IfBOOL;
	delayToSwitchValve17to16: TOF;
	PT030202realValue: REAL;
	PT030302realValue: REAL;
	PT030402realValue: REAL;
	FIT030302realValue: REAL;
	F_P030602: PID;
	P_P030602: PID;
	FIT030202realValue: REAL;
	QIT030102realValue: REAL;
	freqP030601: LIN_TRAFO;
	freqP030602: LIN_TRAFO;
	pt030102:ControlAI;
	pt030202: ControlAI;
	pt030302: ControlAI;
	pt030402: ControlAI;
	fit0301: ControlAI;
	fit030202: ControlAI;
	qit030102: ControlAI;
	fit030302:ControlAI;
	PT030102alarm: BOOL;		(*авария датчика*)
	PT030202alarm: BOOL;
	PT030302alarm: BOOL;
	PT030402alarm: BOOL;
	FIT0301alarm: BOOL;
	FIT030202alarm: BOOL;
	FIT030302alarm: BOOL;
	QIT030102alarm: BOOL;

	testReal: REAL;
	testReal1: REAL;
	testReal2: REAL;
	testBool1: BOOL;
	testBool2: BOOL;
	toNextStartP030201timer: WORD;
	toNextStartP030202timer: WORD;


	PT0303setValue: REAL;		(*Задание максимального давления на РТ03.03*)

	alarmP030101: BOOL;
	alarmP030102: BOOL;
	testBOOL: BOOL;
	testUINT: UINT;
	testTime: TIME;
	testUIN: UDINT;
	BMTflowToCascade: REAL;		(*Расход в БМТ, от которого рассчитываются уставки расхода
			осмосов 1 и 2, каскадно.*)
	isCascade: BOOL;		(*0 = уставка расходу своя, не каскад
			1 = уставка каскадная от расхода БМТ*)
	OPAN_realStub: WORD;
	OPANboolStub: BOOL;
	OPANsetWordP0301: WORD;		(*****************удалить когда пропишешь переменные удаленной панели*********************************)
	OPANwriteSetWord: WORD;		(************************************************удали когда пропишешь переменные удаленной панели*************************************)
	OPANsetWordP0302: WORD;		(***************************удали после того как пропишешь переменные удаленной панели********************************************)
	OPANsetWordOsmos: WORD;		(********************************удали когда пропишешь переменные удаленной панели********************************)

	onStartCatcher: R_TRIG;

	tof1: TOF;
	tof2: TOF;
	tof3: TOF;
	tof4: TOF;
	tof5: TOF;
	tof6: TOF;
	setWordP0301: WORD;		(*конфигурация работы Р0301*)
	setWordP0302: WORD;		(*Конфигурация работы доз.насосов Р03.01*)
	setWordOsmos: WORD;		(*Конфигурация режимов работы осмосов*)
	cascadeTrig: RS;
	setCascadeOnStart: IfBOOL;
END_VAR
VAR RETAIN
	counterP030101: DWORD;		(*счетчик включений насоса Р03.01/01*)
	counterP030102: DWORD;		(*счетчик включений насоса Р03.01/02*)
	daysOfWorkP030101: WORD;		(*количество дней работы насоса Р03.01/01*)
	daysOfWorkP030102: WORD;		(*количество дней работы насоса Р03.01/02*)
	hoursOfWorkP030101: WORD;		(*количество часов работы насоса Р03.01/01*)
	hoursOfWorkP030102: WORD;		(*количество часов работы насоса Р03.01/02*)
	minutesOfWorkP030101: WORD;		(*количество минут работы Р03.01/01*)
	minutesOfWorkP030102: WORD;		(*количество минут работы насоса Р03.01/02*)
	secondsOfWorkP030101: WORD;		(*количество секунд работы насоса Р03.01/01*)
	secondsOfWorkP030102: WORD;		(*количество секунд работы насоса Р03.01/02*)

	counterP030201: DWORD;
	counterP030202: DWORD;
	daysOfWorkP030201: WORD;
	daysOfWorkP030202: WORD;
	hoursOfWorkP030201: WORD;
	hoursOfWorkP030202: WORD;
	minutesOfWorkP030201: WORD;
	minutesOfWorkP030202: WORD;
	secondsOfWorkP030202: WORD;

	counterOsmos1: DWORD;
	counterOsmos2: DWORD;
	daysOfWorkOsmos1: WORD;
	hoursOfWorkOsmos1: WORD;
	minutesOfWorkOsmos1: WORD;
	secondsOfWorkOsmos1: WORD;
	daysOfWorkOsmos2: WORD;
	hoursOfWorkOsmos2: WORD;
	secondsOfWorkP030201: WORD;
	statWordP0301: WORD;		(*статусы состояния насосов Р03.01*)
	statWordP0302: WORD;		(*Статусы состояния доз.насосов Р03.02 на входе осмос 2.*)
	statWordOsmos: WORD;		(*статус состояни осмосов*)
	setWordP0301onStart: WORD;
	setWordP0302onStart: WORD;
	setWordOsmosOnStart: WORD;
	isCascadeOnStart: BOOL;
	FIT0303_SetCascade: REAL;
	PT0301startValue: REAL;		(*Давление РТ0301 для запуска насоса*)
	FIT0303setValue: REAL;		(*Задание расхода для осмоса*)
	PT0302setMaxValue: REAL;
	PT0303setMaxValue: REAL;		(*Задание максимального давления на РТ03.03*)
	PT0304setMaxValue: REAL;
	KP_F_P030601: REAL := 1;
	I_F_P030601: REAL := 10;
	D_F_P030601: REAL := 1;
	KP_P_P030601: REAL := 1;
	I_P_P030601: REAL := 10;
	D_P_P030601: REAL := 1;
	KP_F_P030602: REAL := 1;
	I_F_P030602: REAL := 10;
	D_F_P030602: REAL := 1;
	KP_P_P030602: REAL := 1;
	I_P_P030602: REAL := 10;
	D_P_P030602: REAL := 1;
	setMaxPumpDosingValueP0302: REAL;		(*задание максимальной производительности доз.насоса, в мл/мин*)
	setKoeffProportionalityP0302: REAL;		(*Задание мл на кубометр (коэф.пропорциональности между расходом и дозированием)*)
	CHECKING_DELAY_TIME: TIME;		(*время задержки начала контроля параметра (например, задержка
			контроля эк.манометра после насоса, время на разгон).*)
	DELAY_REPEATED_START_SEC: WORD;		(*время задержки повторного пуска насосов, сек, защита от частых пусков*)
	DELAY_TO_OFF_VALVE: TIME;
	DELAY_TO_CHECK_PT0301: TIME;
	DELAY_TO_SWITCH_VALVE: TIME;		(*время задержки до переключения клапанов после запуска насоса Р0306*)
	DELAY_TO_CLOSE_VALVE: TIME;		(*задержка до начала закрытия клапанов после выключения насосов*)
	FIT0301maxValue: REAL;
	FIT030201maxValue: REAL;
	FIT030301maxValue: REAL;
	FIT030202maxValue: REAL;
	FIT030302maxValue: REAL;
	QIT030101maxValue: REAL;
	QIT030102maxValue: REAL;
	PT030101maxValue: REAL;		(*Максимальное значение показаний датчика РТ03.01/01
			(при 20мА)*)
	PT030201maxValue: REAL;
	PT030301maxValue: REAL;
	PT030401maxValue: REAL;
	PT030102maxValue: REAL;
	PT030202maxValue: REAL;
	PT030302maxValue: REAL;
	PT030402maxValue: REAL;
END_VAR
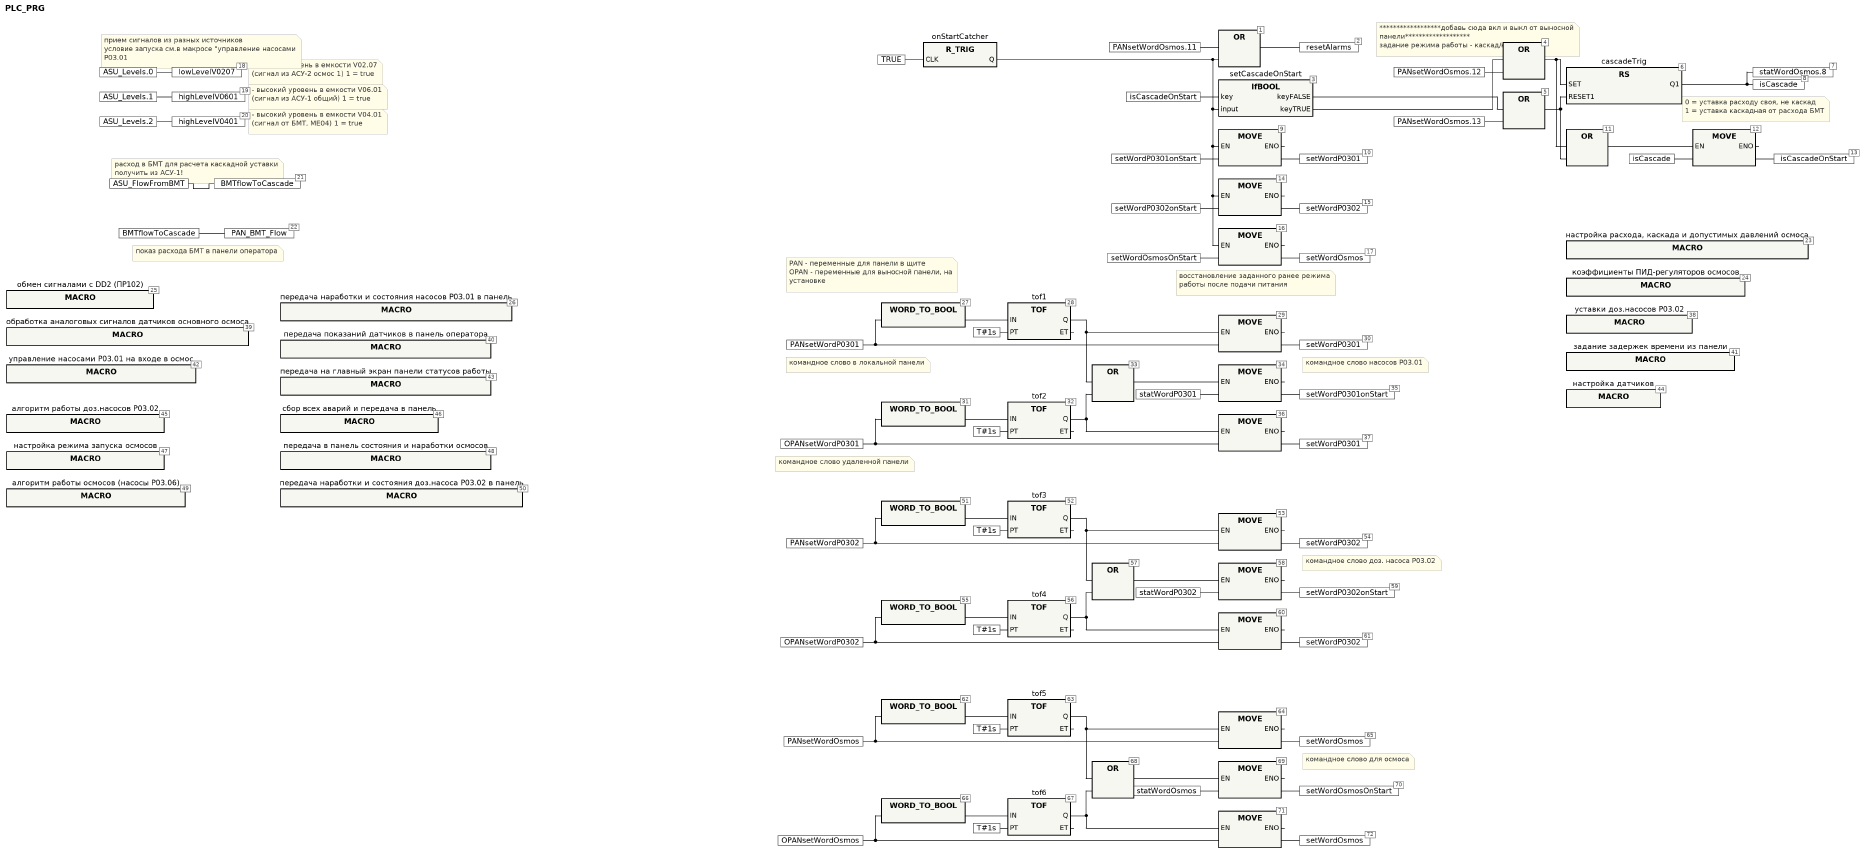
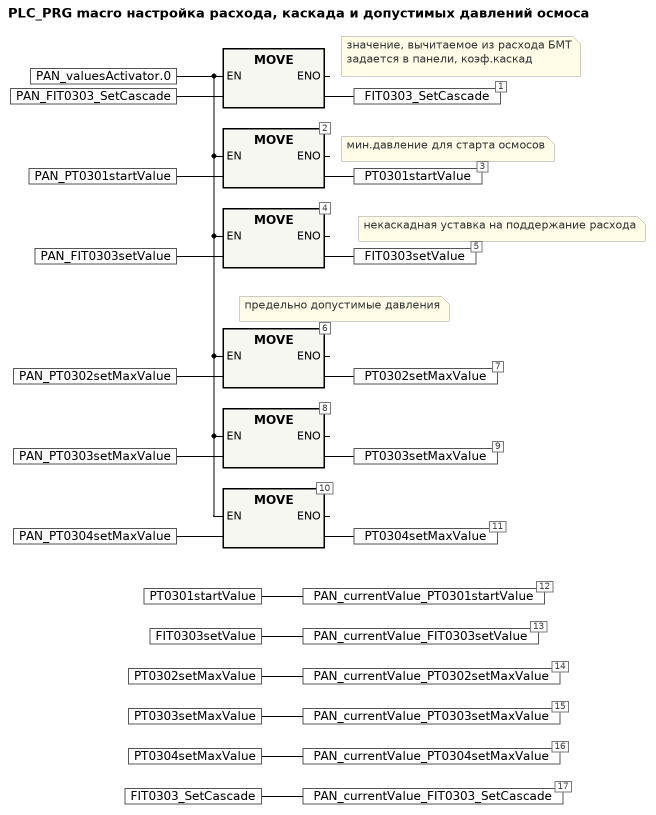
[picture p1: PLC_PRG macro настройка расхода, каскада и допустимых давлений осмоса (CFC)]
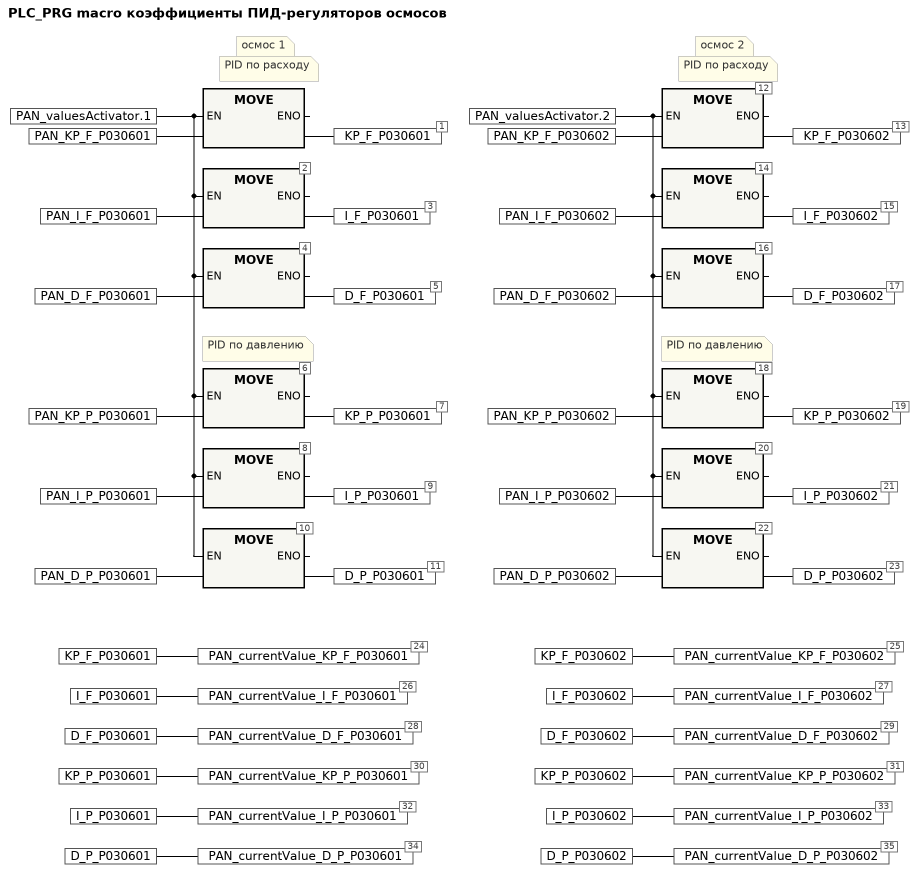
[picture p2: PLC_PRG macro коэффициенты ПИД-регуляторов осмосов (CFC)]
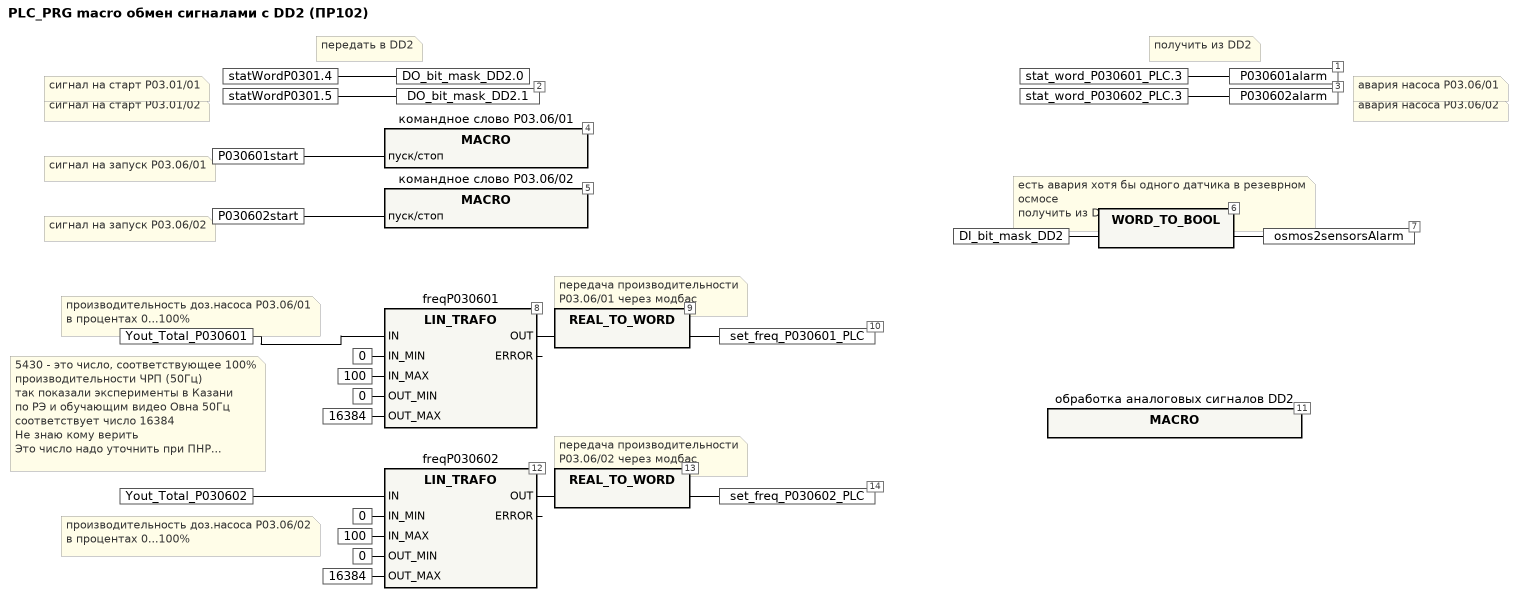
[picture p3: PLC_PRG macro обмен сигналами с DD2 (ПР102) (CFC)]
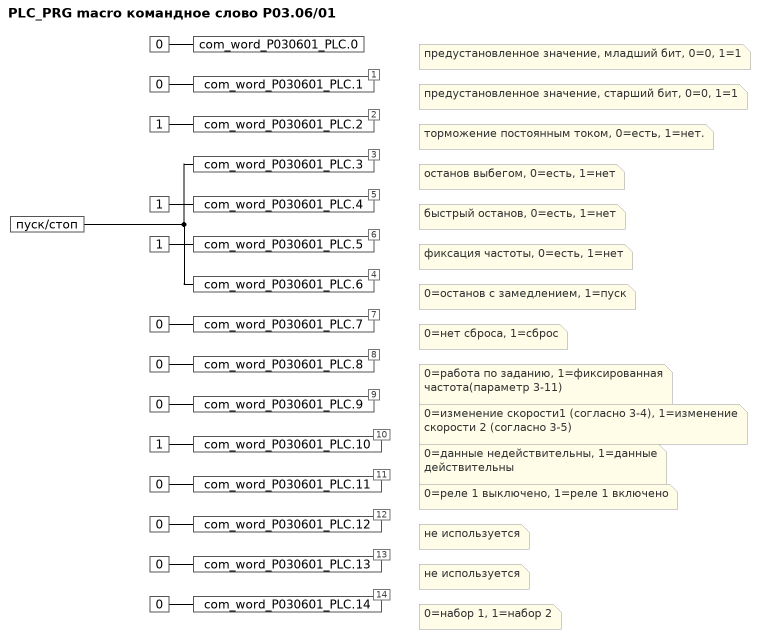
[picture p4: PLC_PRG macro командное слово Р03.06/01 (CFC)]
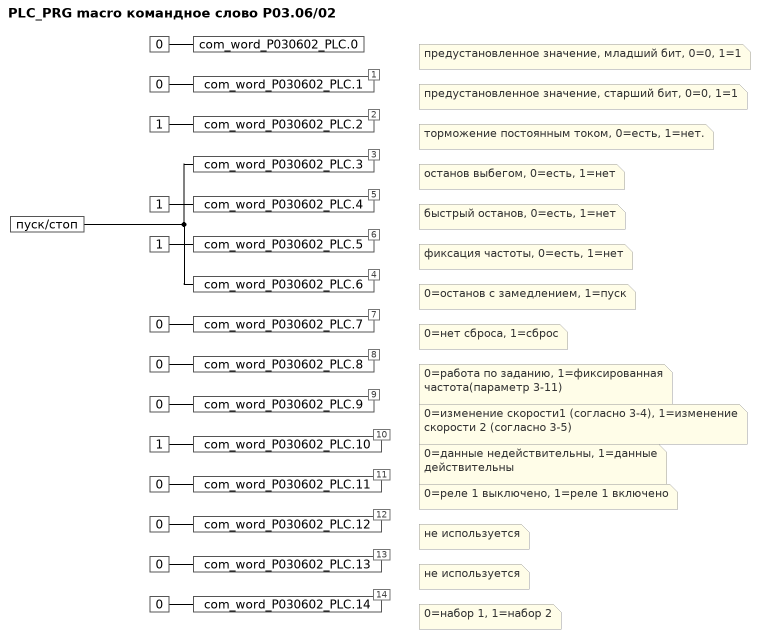
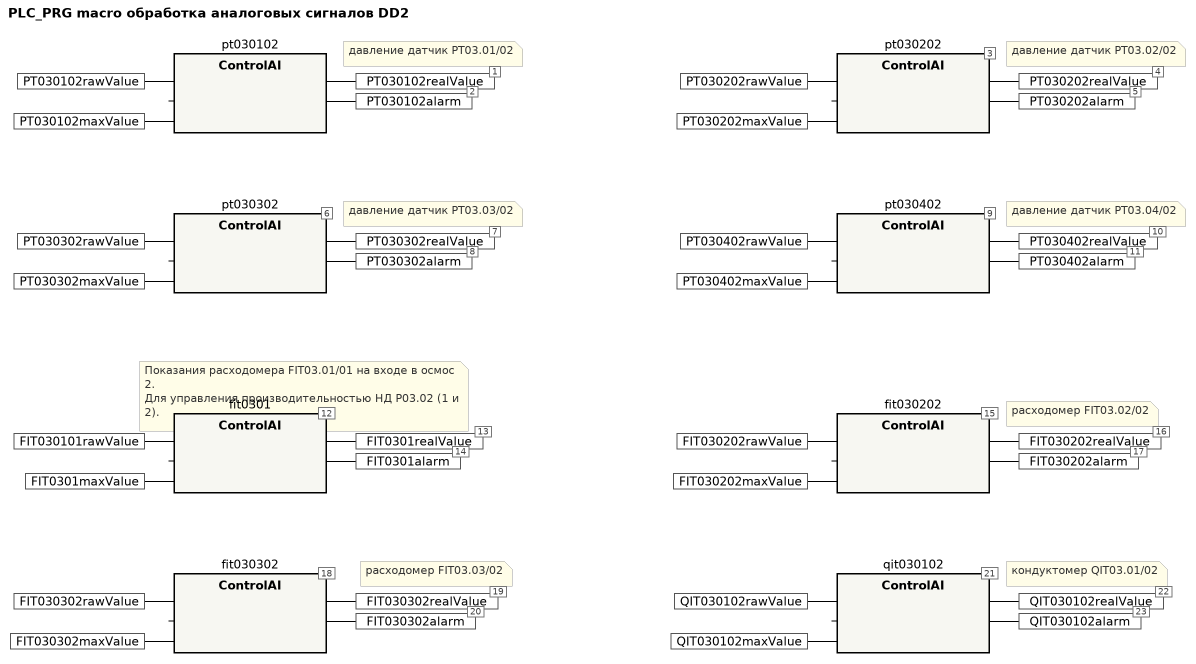
[picture p6: PLC_PRG macro обработка аналоговых сигналов DD2 (CFC)]
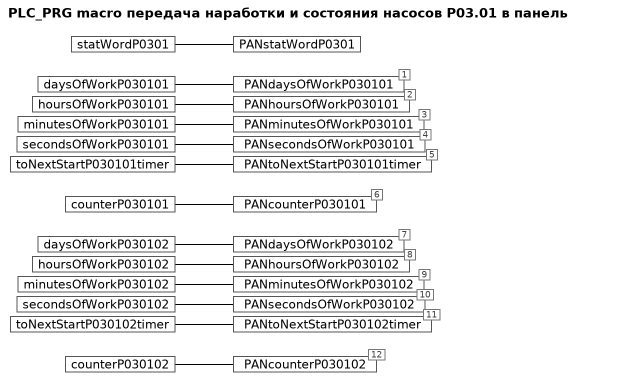
[picture p7: PLC_PRG macro передача наработки и состояния насосов Р03.01 в панель (CFC)]
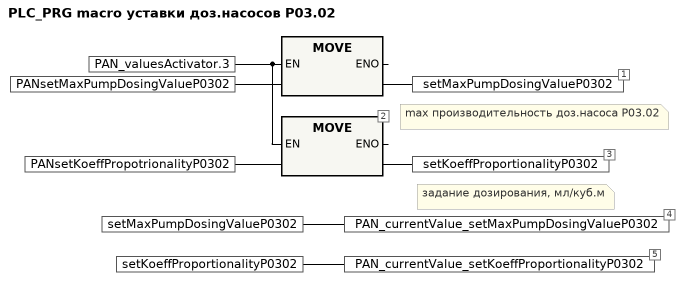
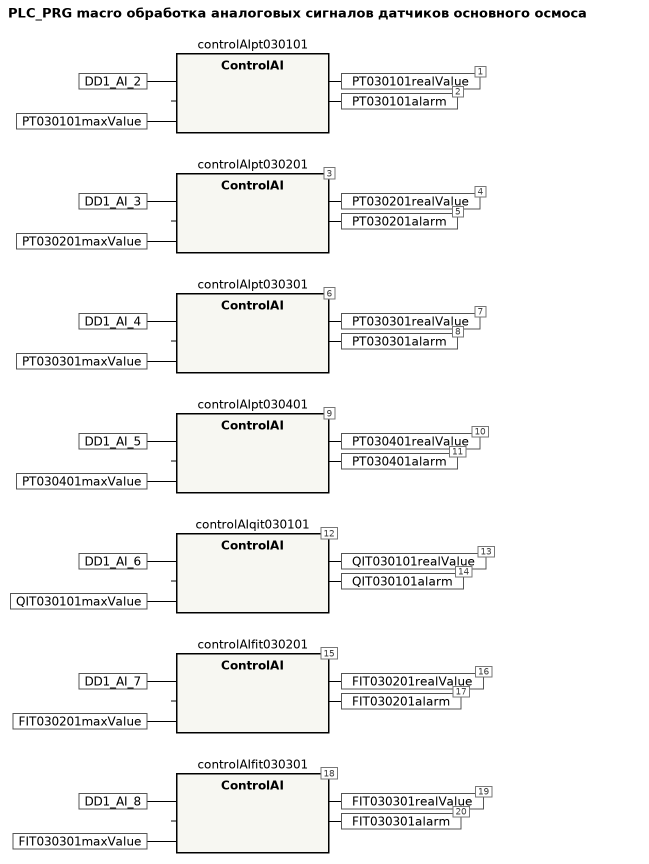
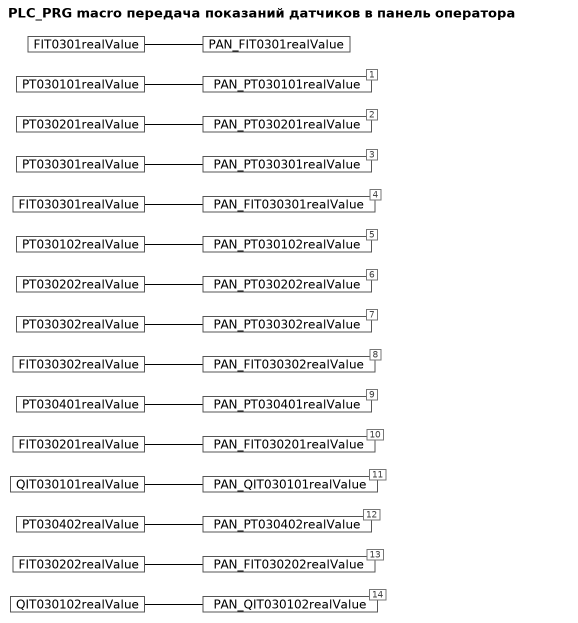
[picture p10: PLC_PRG macro передача показаний датчиков в панель оператора (CFC)]
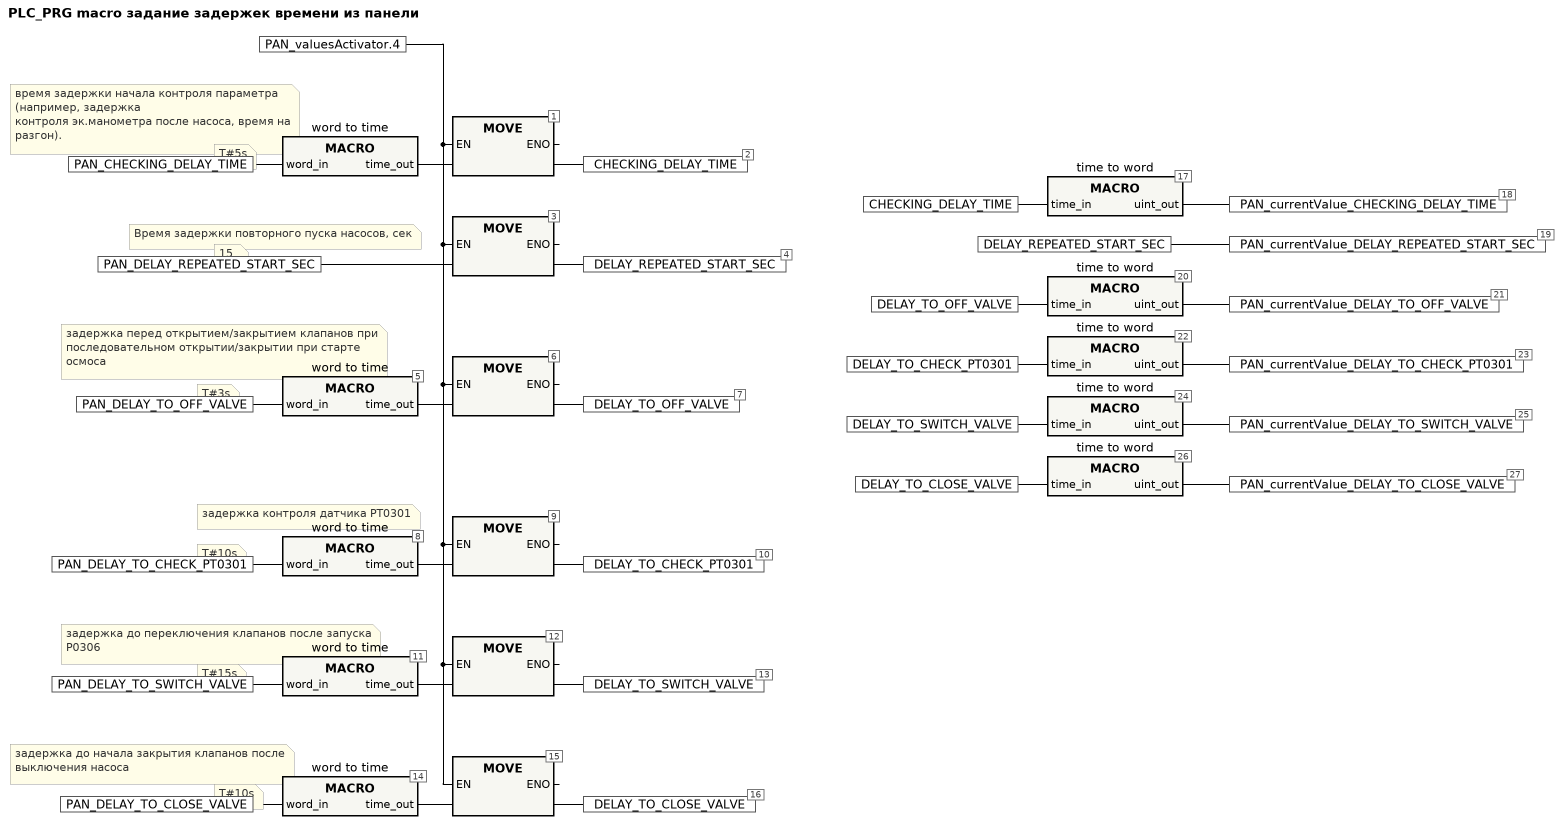
[picture p11: PLC_PRG macro задание задержек времени из панели (CFC)]
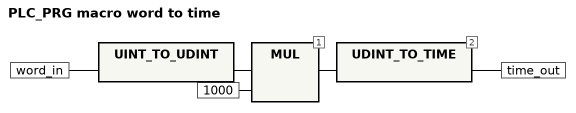
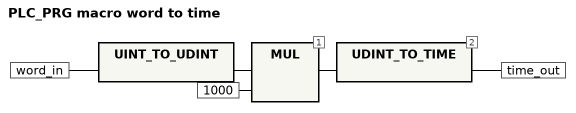
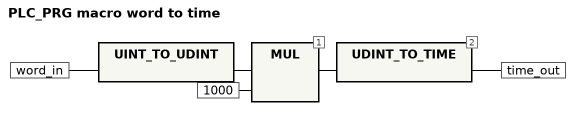
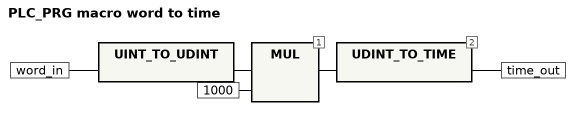
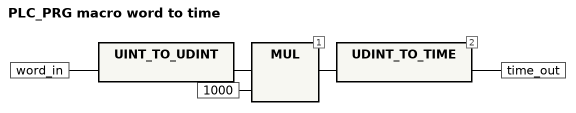
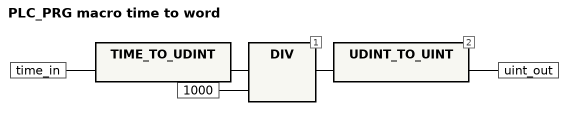
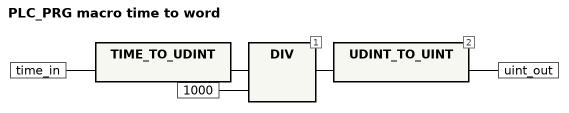
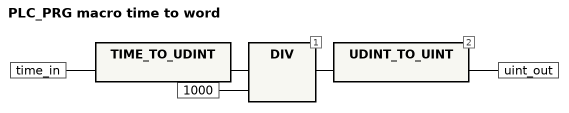
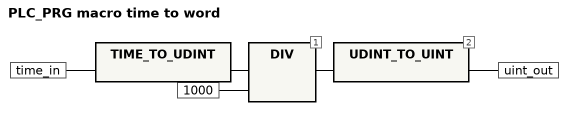
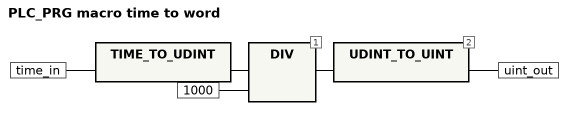
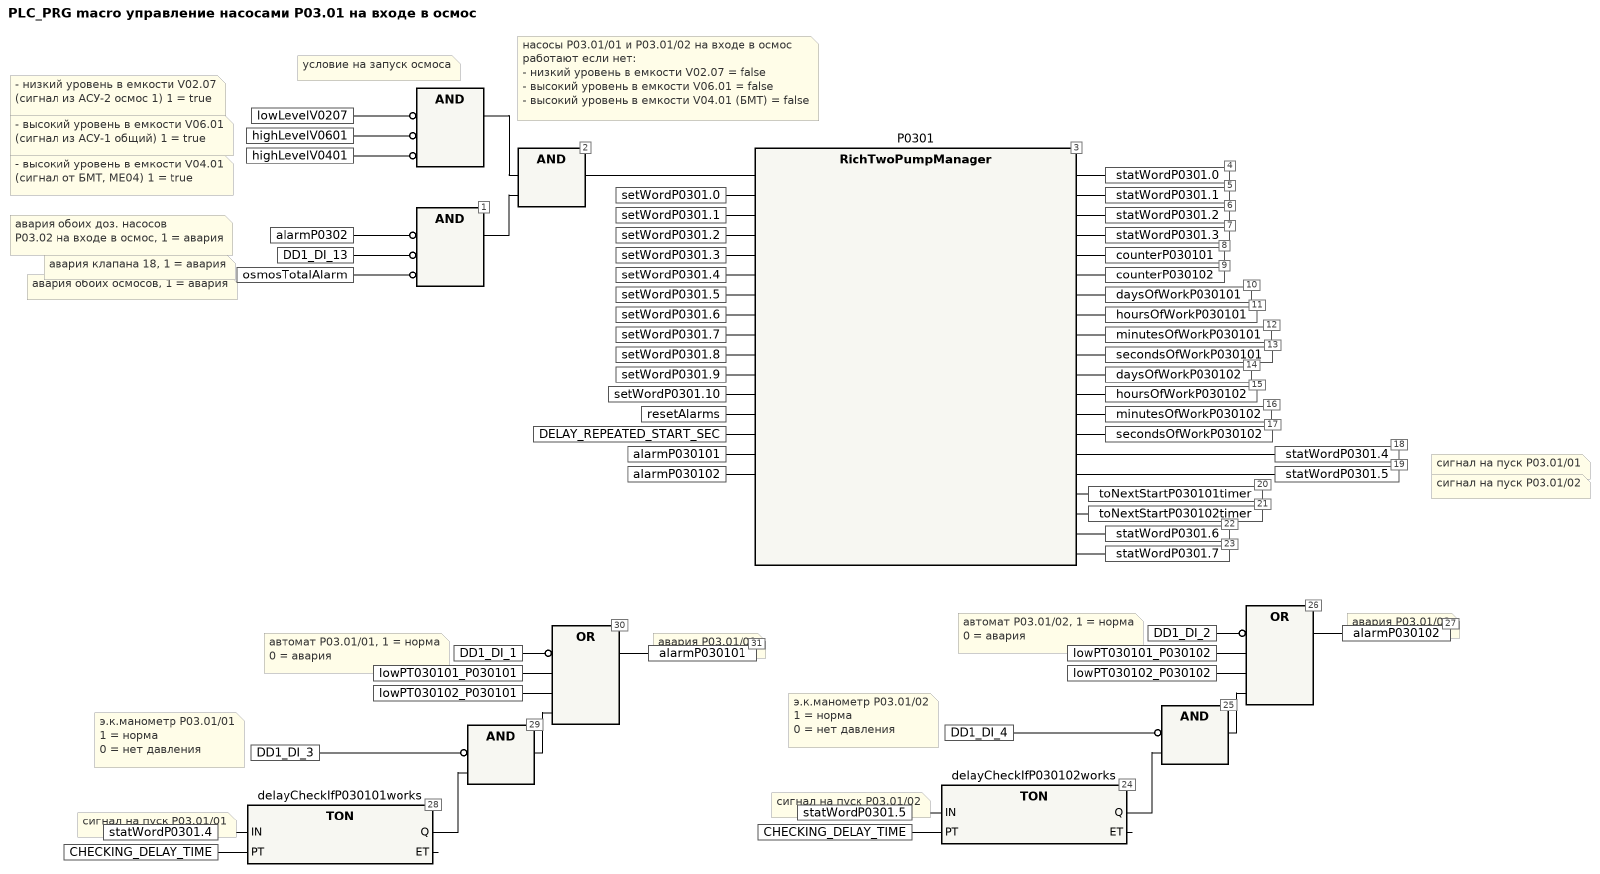
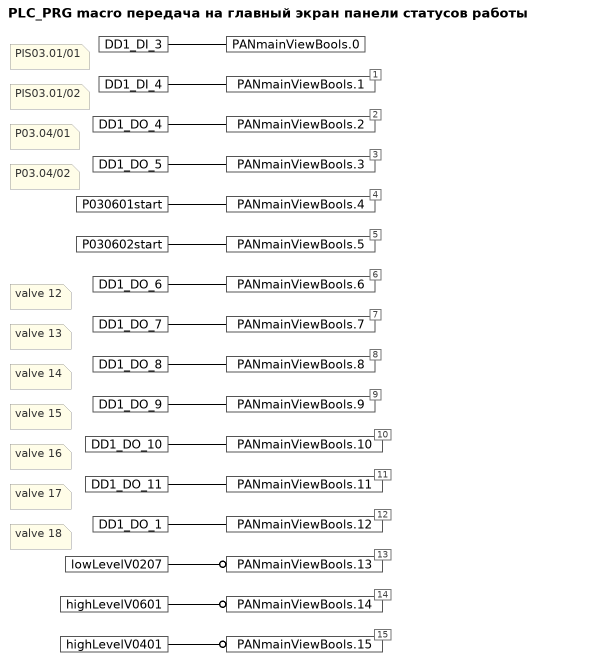
[picture p23: PLC_PRG macro передача на главный экран панели статусов работы (CFC)]
